// TIA Portal project "AUTO-5_UNLOADING_V15.1" (V15.1)

(* hardware
DEVICE "S7-1200 station_1"  S7-1200 Station
   slot 0: "Rack_0"  Rack  V1.0
   slot 1: "PLC_1"  CPU 1214C DC/DC/DC  6ES7 214-1AG40-0XB0  V4.2
   slot 2: "DI 16/DQ 16x24VDC_1"  6ES7 223-1BL32-0XB0  V2.0
   slot 3: "DI 16/DQ 16x24VDC_2"  6ES7 223-1BL32-0XB0  V2.0
DEVICE "HMI_1"  KTP700 Basic PN
   slot 0: "HMI_1"  KTP700 Basic PN  6AV2 123-2GB03-0AX0  15.1.0.0
   slot 1: "HMI_RT_1"  KTP700 Basic PN  6AV2 123-2GB03-0AX0  15.1.0.0
   slot 5: "HMI_1.IE_CP_1"  PROFINET Interface  15.0.1.0
      slot 1: "PROFINET Interface_1"  PROFINET Interface
         slot 1: "Port_1"  Port
DEVICE "GSD device"  GSD.Device.PN
   slot 0: "Rack"  Rack  V1.0
   slot 0: "CTEU-PN_1"  CTEU-PN  2201471  V1.0.0
      slot 0: "CTEU-PN"  CTEU-PN
      slot 1: "PN-IO Interface"  PN-IO Interface
         slot 1: "Port 1"  Port 1
         slot 2: "Port 2"  Port 2
   slot 1: "VAEM-L1-S-8-PT_1"  VAEM-L1-S-8-PT  573384
      slot 0: "VAEM-L1-S-8-PT"  VAEM-L1-S-8-PT
*)

// ===== PLC "PLC_1"  CPU 1214C DC/DC/DC =====

VAR_GLOBAL   // PLC tag table "Default tag table"
   "AUTO_ON_PB" AT %I0.6 : Bool;
   "AUTO_OFF_PB" AT %I0.7 : Bool;
   "CONTROL_OFF" AT %I0.1 : Bool;
   "AUTO_MODE" AT %I0.4 : Bool;
   "MANUAL_MODE" AT %I0.5 : Bool;
   "FAULT RESET" AT %I0.3 : Bool;
   "AIR PRESSURE SWITCH" AT %I1.1 : Bool;
   "PLUG_COUNT" AT %I1.2 : Bool;
   "Tag_14" AT %I1.3 : Bool;
   "Tag_15" AT %I1.4 : Bool;
   "Tag_16" AT %I1.5 : Bool;
   "Tag_17" AT %I2.0 : Bool;
   "Tag_19" AT %I2.2 : Bool;
   "INDIVIDULISER_DOWN" AT %I2.4 : Bool;
   "Tag_18" AT %I2.1 : Bool;
   "INDIVIDULISER_UP" AT %I2.3 : Bool;
   "TRAY LIFTING HEIGHT LEVELING_UP" AT %I2.5 : Bool;
   "TRAY LIFTING HEIGHT LEVELING_DOWN" AT %I2.6 : Bool;
   "TRAY LIFTING CYLINDER _UP" AT %I2.7 : Bool;
   "TRAY LIFTING CYLINDER _DOWN" AT %I3.0 : Bool;
   "TRAY LIFTING CYLINDER_FORWARD_RS" AT %I3.1 : Bool;
   "TRAY LIFTING CYLINDER_REVERSE_RS" AT %I3.2 : Bool;
   "PLUG LIFTING CYLINDER_UP" AT %I3.4 : Bool;
   "PLUG LIFTING CYLINDER_DOWN" AT %I3.3 : Bool;
   "PLUG LIFTING CYLINDER_FORWARD" AT %I3.5 : Bool;
   "PLUG LIFTING CYLINDER_REVERSE" AT %I3.6 : Bool;
   "TRAY STOPPER_UP" AT %I4.0 : Bool;
   "Tag_33" AT %I3.7 : Bool;
   "MPCB_TRIPPED" AT %I0.0 : Bool;
   "PLUG SENSOR MOUNTED ON CHUTE_INPUT" AT %I1.0 : Bool;
   "TRAY_PRESENT LEFT" AT %I4.7 : Bool;
   "TRAY RIGHT SENSOR" AT %I4.1 : Bool;
   "Tag_40" AT %I5.2 : Bool;
   "TRAY LEFT SENSOR" AT %I5.0 : Bool;
   "Tag_42" AT %I5.5 : Bool;
   "UPPER CONVEYOR LEFT  SENSOR" AT %I4.4 : Bool;
   "UPPER CONVEYOR RIGHT SENSOR" AT %I4.3 : Bool;
   "TRAY_PRESENT_RIGHT" AT %I4.5 : Bool;
   "WALKER BEAM UP" AT %Q0.0 : Bool;
   "WALKER BEAM DOWN" AT %Q0.1 : Bool;
   "Tag_12" AT %Q1.0 : Bool;
   "Tag_13" AT %Q1.1 : Bool;
   "CYCLE STRT ILPB INDICATOR" AT %Q0.3 : Bool;
   "PLUG_LIFT_DOWN" AT %Q6.0 : Bool;
   "PLUG LIFTING CYLINDER UP(1)" AT %Q6.1 : Bool;
   "GRIPPER_HOLD" AT %Q6.2 : Bool;
   "Tag_49" AT %Q7.4 : Bool;
   "TRAY PICKUP HEIGHT DOWN" AT %Q7.0 : Bool;
   "TRAY PICKUP UP" AT %Q7.1 : Bool;
   "TRAY LIFTING DOWN" AT %Q6.6 : Bool;
   "TRAY LIFTING CYLINDER  UP_OUTPUT" AT %Q6.7 : Bool;
   "TRAY LIFTING FWD_" AT %Q7.2 : Bool;
   "TRAY_LIFT_REVERSE" AT %Q7.3 : Bool;
   "PLUG_LIFT_REV" AT %Q6.4 : Bool;
   "PLUG_LIFT_FWD" AT %Q6.5 : Bool;
   "Tag_58" AT %Q7.6 : Bool;
   "Tag_59" AT %Q7.7 : Bool;
   "Tag_60" AT %Q7.5 : Bool;
   "AUTO CYCLE ON- YELLOW LAMP" AT %Q5.3 : Bool;
   "Tag_62" AT %Q5.4 : Bool;
   "ALL UNIT INITIAL- GREEN LAMP" AT %Q5.5 : Bool;
   "Tag_64" AT %Q0.6 : Bool;
   "FB_SENSOR OUTPUT" AT %Q5.6 : Bool;
   "RED LAMP" AT %Q5.7 : Bool;
   "GRIPPER_UNHOLD" AT %Q6.3 : Bool;
   "CONVEYOR -1 RUN FROM HMI" AT %M100.0 : Bool;
   "CONVEYOR -1 RUN OUTPUT" AT %M150.0 : Bool;
   "CONVEYOR 2 RUN FROM HMI" AT %M100.1 : Bool;
   "Tag_2" AT %M100.2 : Bool;
   "EMERGENCY" AT %M100.3 : Bool;
   "CYCLE START" AT %M100.4 : Bool;
   "CYCLE STOP" AT %M100.5 : Bool;
   "RESET" AT %M100.6 : Bool;
   "CONTROL ON" AT %M100.7 : Bool;
   "AUTO MODE" AT %M101.0 : Bool;
   "MANUAL MODE" AT %M101.1 : Bool;
   "AIR PRESSURE" AT %M101.2 : Bool;
   "PLUG SENSOR MOUNTED ON CHUTE" AT %M101.3 : Bool;
   "PLUG COUNTING" AT %M101.4 : Bool;
   "INDIVIDULISER-1 UP READ SWITCH" AT %M101.5 : Bool;
   "INDIVIDULISER-1 DOWN READ SWITCH" AT %M101.6 : Bool;
   "INDIVIDULISER -2 UP RS" AT %M101.7 : Bool;
   "INDIVIDULISER -2 DOWN RS" AT %M102.0 : Bool;
   "INDIVIDULISER -3 UP  RS" AT %M102.1 : Bool;
   "INDIVIDULISER -3 DOWN RS" AT %M102.2 : Bool;
   "INDIVIDULISER -4 UP RS" AT %M102.3 : Bool;
   "INDIVIDULISER -4 DOWN RS" AT %M102.4 : Bool;
   "TRAY LIFTING HEIGHT LEVELING UP READ SWITCH" AT %M102.5 : Bool;
   "TRAY LIFTING HEIGHT LEVELING DOWN READ SWITCH" AT %M102.6 : Bool;
   "TRAY LIFTING CYLINDER  UP  READ SWITCH" AT %M102.7 : Bool;
   "TRAY LIFTING CYLINDER DOWN READ SWITCH" AT %M103.0 : Bool;
   "TRAY LIFTING CYLINDER FORWARD READ SWITCH" AT %M103.1 : Bool;
   "TRAY LIFTING CYLINDER REVERSE READ SWITCH" AT %M103.2 : Bool;
   "PLUG LIFTING CYLINDER UP READ SWITCH" AT %M103.3 : Bool;
   "PLUG LIFTING CYLINDER DOWN READ SWITCH" AT %M103.4 : Bool;
   "PLUG LIFTING CYLINDER FORWARD READ SWITCH" AT %M103.5 : Bool;
   "PLUG LIFTING CYLINDER REVERSE READ SWITCH" AT %M103.6 : Bool;
   "TRAY STOPPER UP READ SWITCH" AT %M103.7 : Bool;
   "TRAY STOPPER DOWN READ SWITCH" AT %M104.0 : Bool;
   "TRAY LATCH UP READ SWITCH" AT %M104.1 : Bool;
   "TRAY LATCH DOWN READ SWITCH" AT %M104.2 : Bool;
   "CONVEYOR -1 MPCB TRIP" AT %M104.3 : Bool;
   "CONVEYOR -2 MPCB TRIP" AT %M104.4 : Bool;
   "INDIVIDUAL CYLINDER UP FROM HMI" AT %M104.5 : Bool;
   "INDIVIDUAL CYLINDER DOWN FROM HMI" AT %M104.6 : Bool;
   "TRAY LIFTING HEIGHT LEVELING UP FROM HMI" AT %M104.7 : Bool;
   "TRAY LIFTING HEIGHT LEVELING DOWN FROM HMI" AT %M105.0 : Bool;
   "TRAY LIFTING CYLINDER  UP FROM HMI" AT %M105.1 : Bool;
   "TRAY LIFTING CYLINDER  DOWN FROM HMI" AT %M105.2 : Bool;
   "TRAY LIFTING CYLINDER FORWARD FROM HMI" AT %M105.3 : Bool;
   "TRAY LIFTING CYLINDER REVERSE FROM HMI" AT %M105.4 : Bool;
   "PLUG LIFTING CYLINDER UP FROM HMI" AT %M105.5 : Bool;
   "PLUG LIFTING CYLINDER  DOWN FROM HMI" AT %M105.6 : Bool;
   "PLUG LIFTING CYLINDER FORWARD FROM HMI" AT %M105.7 : Bool;
   "CONVEYOR 2 RUN OUTPUT" AT %M150.1 : Bool;
   "INDIVIDULISER CYLINDER  UP" AT %M150.2 : Bool;
   "INDIVIDULISER CYLINDER DOWN" AT %M150.3 : Bool;
   "TRAY LIFTING HEIGHT LEVELING UP" AT %M150.4 : Bool;
   "TRAY LIFTING HEIGHT LEVELING DOWN" AT %M150.5 : Bool;
   "TRAY LIFTING CYLINDER  UP" AT %M150.6 : Bool;
   "TRAY LIFTING CYLINDER  DOWN" AT %M150.7 : Bool;
   "TRAY LIFTING CYLINDER FORWARD" AT %M151.0 : Bool;
   "TRAY LIFTING CYLINDER REVERSE" AT %M151.1 : Bool;
   "PLUG LIFTING CYLINDER UP" AT %M151.2 : Bool;
   "PLUG LIFTING CYLINDER DOWN" AT %M151.3 : Bool;
   "PLUG LIFTING CYLINDER FORWARD" AT %M151.4 : Bool;
   "PLUG LIFTING CYLINDER REVERSE" AT %M151.5 : Bool;
   "TRAY STOPPER UP" AT %M151.6 : Bool;
   "TRAY STOPPER DOWN" AT %M151.7 : Bool;
   "TRAY LATCH UP" AT %M152.0 : Bool;
   "TRAY LATCH DOWN" AT %M152.1 : Bool;
   "INITIAL CONDITION ON LAMP" AT %M152.2 : Bool;
   "TOWER LAMP RED" AT %M152.3 : Bool;
   "TOWER LAMP YELLOW" AT %M152.4 : Bool;
   "TOWER LAMP GREEN" AT %M152.5 : Bool;
   "BUZZER" AT %M152.6 : Bool;
   "PLUG LIFTING CYLINDER REVERSE FROM HMI" AT %M106.0 : Bool;
   "TRAY STOPPER UP FROM HMI" AT %M106.1 : Bool;
   "TRAY STOPPER DOWN FROM HMI" AT %M106.2 : Bool;
   "TRAY LATCH UP FROM HMI" AT %M106.3 : Bool;
   "TRAY LATCH DOWN FROM HMI" AT %M106.4 : Bool;
   "CYCLE START FLAG" AT %M200.0 : Bool;
   "ALL INDIVIDULISER UP RS" AT %M200.1 : Bool;
   "ALL INDIVIDULISER DOWN RS" AT %M200.2 : Bool;
   "Clock_Byte" AT %MB0 : Byte;
   "Clock_10Hz" AT %M0.0 : Bool;
   "Clock_5Hz" AT %M0.1 : Bool;
   "Clock_2.5Hz" AT %M0.2 : Bool;
   "Clock_2Hz" AT %M0.3 : Bool;
   "Clock_1.25Hz" AT %M0.4 : Bool;
   "Clock_1Hz" AT %M0.5 : Bool;
   "Clock_0.625Hz" AT %M0.6 : Bool;
   "Clock_0.5Hz" AT %M0.7 : Bool;
   "System_Byte" AT %MB1 : Byte;
   "FirstScan" AT %M1.0 : Bool;
   "DiagStatusUpdate" AT %M1.1 : Bool;
   "AlwaysTRUE" AT %M1.2 : Bool;
   "AlwaysFALSE" AT %M1.3 : Bool;
   "TRAY PRESENT SENSOR-LEFT PROXIMITY" AT %M106.5 : Bool;
   "TRAY PRESENT SENSOR-RIGHT PROXIMITY" AT %M106.6 : Bool;
   "TRAY PRESENT SENSOR BEFORE-LEFT PROXIMITY(1)" AT %M106.7 : Bool;
   "TRAY PRESENT BEFORE SENSOR-RIGHT PROXIMITY(1)" AT %M107.0 : Bool;
   "CONVEYOR -1 STOP FROM HMI" AT %M107.1 : Bool;
   "CONVEYOR -2 STOP FROM HMI" AT %M107.2 : Bool;
   "PLUG COUNTING PULSE" AT %M50.0 : Bool;
   "PLUG COUNTING RESET" AT %M50.1 : Bool;
   "Tag_36" AT %M30.0 : Bool;
   "TRAY LIFTING CYLINDER  DOWN_TRIGGER" AT %M30.1 : Bool;
   "Tag_43" AT %M25.0 : Bool;
   "Tag_44" AT %M20.0 : Bool;
   "Tag_46" AT %M10.1 : Bool;
   "TOWER LAMP BLUE" AT %M152.7 : Bool;
   "TOWER LAMP WHITE" AT %M153.0 : Bool;
   "PLUG HOLD FROM HMI" AT %M107.3 : Bool;
   "PLUD UNHOLD FROM HMI" AT %M107.4 : Bool;
   "PLUG HOLD O/P" AT %M153.1 : Bool;
   "PLUG UNHOLD O/P" AT %M153.2 : Bool;
   "TRIGGER_RESET_PLUG_COUNT" AT %M15.0 : Bool;
   "Tag_69" AT %M15.1 : Bool;
   "Tag_70" AT %M15.2 : Bool;
   "Tag_71" AT %M9.0 : Bool;
   "Tag_72" AT %M9.1 : Bool;
   "Tag_73" AT %M22.0 : Bool;
   "Tag_74" AT %M22.2 : Bool;
   "Tag_75" AT %M22.3 : Bool;
   "Tag_76" AT %M23.0 : Bool;
   "Tag_77" AT %M23.1 : Bool;
   "Tag_78" AT %M24.0 : Bool;
   "Tag_79" AT %M24.2 : Bool;
   "Tag_81" AT %M26.2 : Bool;
   "Tag_82" AT %M24.4 : Bool;
   "Tag_83" AT %M24.6 : Bool;
   "down tray present by pass on" AT %M25.5 : Bool;
   "delay 2s" AT %M40.0 : Bool;
   "1s delay for pallet sensors" AT %M40.2 : Bool;
   "DELAY 2S FOR DOWN FWD" AT %M40.4 : Bool;
   "Tag_84" AT %M99.0 : Bool;
   "DOWN B" AT %M90.1 : Bool;
   "Tag_41" AT %M90.2 : Bool;
   "Tag_47" AT %M90.7 : Bool;
   "UP B" AT %M90.5 : Bool;
   "INITIAL RESET" AT %I0.2 : Bool;
   "CONTROL ON OUTPUT" AT %Q0.7 : Bool;
   "Tag_7" AT %M15.5 : Bool;
   "Tag_39" AT %M16.3 : Bool;
   "Tag_85" AT %M16.5 : Bool;
   "INTER LOCK BIT TAKING UP/DOWN TRAY" AT %M17.2 : Bool;
   "Tag_87" AT %M17.4 : Bool;
   "Tag_1" AT %M16.1 : Bool;
   "Tag_3" AT %M16.2 : Bool;
   "PLUG PRESENT SENSOR AFTER REROLLING" AT %I5.4 : Bool;
   "AUTO WALKER UP" AT %M300.0 : Bool;
   "MAN WALKER UP" AT %M500.0 : Bool;
   "WALKER DOWN" AT %M300.1 : Bool;
   "MAN WALKER DOWN" AT %M500.1 : Bool;
   "Tag_5" AT %M300.2 : Bool;
   "HMI_PLUG_LIFT_UP" AT %M500.2 : Bool;
   "Tag_8" AT %M300.3 : Bool;
   "HMI_PLUG_LIFT_DOWN" AT %M500.3 : Bool;
   "Tag_10" AT %M300.4 : Bool;
   "HMI_GRIPPER_HOLD" AT %M500.4 : Bool;
   "Tag_21" AT %M300.5 : Bool;
   "HMI_GRIPPER_UNHOLD" AT %M500.5 : Bool;
   "Tag_23" AT %M300.6 : Bool;
   "HMI_TRAY_LIFT_DOWN" AT %M500.6 : Bool;
   "Tag_25" AT %M300.7 : Bool;
   "HMI_TRAY_LIFT_UP" AT %M500.7 : Bool;
   "Tag_27" AT %M301.0 : Bool;
   "HMI_TRAY_HEIGHT_DOWN" AT %M501.0 : Bool;
   "Tag_29" AT %M301.1 : Bool;
   "HMI_TRAY_HEIGHT_UP" AT %M501.1 : Bool;
   "Tag_31" AT %M301.2 : Bool;
   "HMI_TRAY_LIFT_FORWARD" AT %M501.2 : Bool;
   "Tag_34" AT %M301.3 : Bool;
   "HMI_TRAY_LIFT_REVERSE" AT %M501.3 : Bool;
   "AUTO ON" AT %M310.0 : Bool;
   "Tag_11" AT %M310.2 : Bool;
   "Tag_53" AT %M310.3 : Bool;
   "25 COUNT REACHED" AT %M310.5 : Bool;
   "Tag_86" AT %M310.7 : Bool;
   "ALL UNIT INITIAL" AT %M310.1 : Bool;
   "CONVY ON BIT" AT %M301.5 : Bool;
   "Tag_90" AT %M302.1 : Bool;
   "Tag_91" AT %M302.0 : Bool;
   "Tag_92" AT %MW300 : Int;
   "Tag_93" AT %MW302 : Int;
   "HMI_PLUG_LIFT_FWD" AT %M502.0 : Bool;
   "HMI_PLUG_LIFT_REV" AT %M502.1 : Bool;
   "Tag_96" AT %M312.0 : Bool;
   "PLUG LIFTING CYL DOWN SETBIT" AT %M600.3 : Bool;
   "PLUG GRIP SETBIT" AT %M600.4 : Bool;
   "Tag_99" AT %M610.5 : Bool;
   "TRAY UP SETBIT" AT %M610.0 : Bool;
   "Tag_101" AT %M610.2 : Bool;
   "PLUG GRIPPER UP CYL SETBIT" AT %M600.5 : Bool;
   "PLUG GRIP REV CYL SETBIT" AT %M600.6 : Bool;
   "PLUG LIFTING CYL DOWN  SETBIT" AT %M600.7 : Bool;
   "Tag_105" AT %M601.7 : Bool;
   "PLUG UNGRIP SETBIT" AT %M601.0 : Bool;
   "PLUG LIFTING UP CYL SETBIT" AT %M601.1 : Bool;
   "PLUG LIFTING FWD CYL SETBIT" AT %M601.2 : Bool;
   "Tag_109" AT %MW600 : Int;
   "Tag_110" AT %MW602 : Int;
   "Tag_111" AT %M610.4 : Bool;
   "Tag_112" AT %M610.6 : Bool;
   "TRAY FWD CYL SETBIT" AT %M611.0 : Bool;
   "TRAY DOWN CYL SETBIT" AT %M611.2 : Bool;
   "Tag_115" AT %M611.4 : Bool;
   "Tag_116" AT %M611.6 : Bool;
   "Tag_117" AT %M612.0 : Bool;
   "Tag_118" AT %M612.2 : Bool;
   "Tag_4" AT %MW604 : Int;
   "Tag_68" AT %MW606 : Int;
   "Tag_88" AT %MW610 : Int;
   "Tag_89" AT %MW612 : Int;
   "Tag_97" AT %M601.4 : Bool;
   "Tag_38" AT %M26.0 : Bool;
   "Tag_50" AT %M26.1 : Bool;
   "1s delay for pallet sensors_1" AT %M26.5 : Bool;
   "TRAY LIFTING HEIGHT LEVELING UP_TRIG" AT %M27.0 : Bool;
   "TRAY LIFT CYLINDER FORWARD TRIGGER" AT %M27.4 : Bool;
   "DELAY_2S_TIM" AT %M27.6 : Bool;
   "DELAY 2S FOR DOWN FWD_" AT %M27.7 : Bool;
   "Tag_51" AT %M28.0 : Bool;
   "TRAY LIFTING HEIGHT LEVELING DOWN_TRIGGER" AT %M28.1 : Bool;
   "TRAY LIFTING CYLINDER  UP_TRIGGER" AT %I30.0 : Bool;
   "TRAY LIFTING CYLINDER REVERSE_TRIGGER" AT %M31.0 : Bool;
   "PLUG_COUNT_DISPLAY" AT %MD32 : DInt;
   "SPARE" AT %Q0.5 : Bool;
   "ALL_UNIT_INITIAL" AT %Q0.2 : Bool;
   "Tag_6" AT %M613.0 : Bool;
   "Tag_9" AT %M163.0 : Bool;
   "Tag_20" AT %M163.1 : Bool;
   "Tag_22" AT %M613.1 : Bool;
   "Tag_24" AT %M613.2 : Bool;
   "parts full after rerolling" AT %I5.6 : Bool;
   "RELAY O/P" AT %Q2.0 : Bool;
   "RELAY TRIGGER BIT" AT %M613.6 : Bool;
   "Tag_26" AT %M614.0 : Bool;
   "Tag_28" AT %M614.1 : Bool;
   "ALARM_1" AT %MW60 : Word;
   "ALARM_2" AT %MW62 : Word;
   "Tag_30" AT %M60.0 : Bool;
   "CONTROL OFF" AT %M61.0 : Bool;
   "AUTO_OFF_ERROR" AT %M61.4 : Bool;
   "MPCB_TRIPPED_ERROR" AT %M61.3 : Bool;
   "AIR PRESSURE LOW ERROR" AT %M61.5 : Bool;
   "WAITING FOR PLUGS FROM SB UNIT ERROR" AT %M61.6 : Bool;
   "TRAY NOT  PRESENT ERROR" AT %M61.2 : Bool;
   "Tag_32" AT %M61.1 : Bool;
   "Tag_35" AT %M25.1 : Bool;
   "TRAY NOT PRESENT AT CONVEYOR END" AT %M61.7 : Bool;
   "Tag_45" AT %MW613 : Int;
   "Tag_48" AT %M630.0 : Bool;
   "INITIAL_SEQ_TRIGGER" AT %M110.0 : Bool;
   "TRAY_REVERSE_TRIGGER_INITIAL" AT %M110.1 : Bool;
   "TRAY_HEIGHT_UP_TRIG_INITIAL" AT %M110.2 : Bool;
   "TRAY HEIGHT FORWARD_TRIG_INITIAL" AT %M110.3 : Bool;
   "TRAY HEIGHT DOWN TRIG INITIAL" AT %M110.4 : Bool;
   "Tag_54" AT %MW110 : Int;
   "Tag_37" AT %M111.0 : Bool;
   "Tag_52" AT %M111.1 : Bool;
   "TRAY_HEIGHT_DOWN_INIT" AT %M111.3 : Bool;
   "Tag_55" AT %M112.0 : Bool;
   "Tag_56" AT %M112.1 : Bool;
   "Tag_57" AT %Q0.4 : Bool;
   "AUTO_OFF_TRIGGER_SINGLE CYCLE" AT %M112.2 : Bool;
   "Tag_63" AT %M113.0 : Bool;
   "PLUG TRANSFER SINGLE CYCLE TRIGGER" AT %M115.0 : Bool;
   "HMI_TRAY_PRESENT_INITIAL" AT %M25.2 : Bool;
   "TRAY HEIGHT LIFT INITIAL TRIGGER" AT %M116.0 : Bool;
   "TRAY _LIFT_REVERSE_INITIAL_TRIGGER" AT %M116.1 : Bool;
   "TRAY_LIFT_HEIGHT_DOWN_TRIGGER" AT %M116.2 : Bool;
   "TRAY_LIFT_FWD_INITIAL_TRIGGER" AT %M116.3 : Bool;
   "TRAY_LIFT_DOWN_INITIAL_TRIGGER" AT %M116.4 : Bool;
   "Tag_61" AT %MW115 : Int;
   "DUMMY" AT %M116.7 : Bool;
END_VAR

DATA_BLOCK "RETENTIVES"   // DB3
{ S7_Optimized_Access := 'FALSE' }
VERSION : 0.1
   VAR
      "PLUG COUNTER" : DInt;
      "RESET FLAG" : Bool;
      "PLUG FILLED" : Bool;
      "PLUG DATA" : DInt;
      "15 COUNTS REACH" : Bool;
      "PLUG LIFTING CYLINDER UP READ SWITCH" : Bool;
      "AUTO PLUG HOLD" : Bool;
      "AUTO PLUG UNHOLD" : Bool;
      "PLUG COUNTING RESET" : Bool;
      "ALL INDIVIDULISER DOWN CONFIRM" : Bool;
      "AUTO FWD FLag" : Bool;
      "AUTO REV FLAG" : Bool;
      "ALL INDIVIDULISER DOWN READ SWITCH" : Bool;
      "PLUG LIFTING CYLINDER UP" : Bool;
      "ERROR MSGS MOV BIT" : DInt;
      "ERROR FLAG ON" : Bool;
      "AUTO FWD FLAG DOWN" : Bool;
      "AUTO REV FLAG DOWN" : Bool;
      "AUTO FWD FLAG UP" : Bool;
      "AUTO REV FLAG UP" : Bool;
   END_VAR
BEGIN
END_DATA_BLOCK

// folder: System blocks/Program resources

DATA_BLOCK "PART PRESENT OFF DWELL"   // DB1
{ S7_Optimized_Access := 'TRUE' }
AUTHOR : Simatic
FAMILY : IEC
NAME : IEC_TMR
VERSION : 1.0
// stored: InstanceOfName IEC_TIMER
"IEC_TIMER"
BEGIN
END_DATA_BLOCK

DATA_BLOCK "PARTS COUNT"   // DB2
{ S7_Optimized_Access := 'TRUE' }
AUTHOR : Simatic
FAMILY : IEC
NAME : CNTR
VERSION : 1.0
// stored: InstanceOfName IEC_COUNTER
"IEC_COUNTER"
BEGIN
END_DATA_BLOCK

DATA_BLOCK "WALKER BEAM UP DWELL"   // DB4
{ S7_Optimized_Access := 'TRUE' }
AUTHOR : Simatic
FAMILY : IEC
NAME : IEC_TMR
VERSION : 1.0
// stored: InstanceOfName IEC_TIMER
"IEC_TIMER"
BEGIN
END_DATA_BLOCK

DATA_BLOCK "WALKER DOWN DWELL"   // DB5
{ S7_Optimized_Access := 'TRUE' }
AUTHOR : Simatic
FAMILY : IEC
NAME : IEC_TMR
VERSION : 1.0
// stored: InstanceOfName IEC_TIMER
"IEC_TIMER"
BEGIN
END_DATA_BLOCK

DATA_BLOCK "GRIP DWELL"   // DB6
{ S7_Optimized_Access := 'TRUE' }
AUTHOR : Simatic
FAMILY : IEC
NAME : IEC_TMR
VERSION : 1.0
// stored: InstanceOfName IEC_TIMER
"IEC_TIMER"
BEGIN
END_DATA_BLOCK

DATA_BLOCK "GRIPPER DOWN DWELL"   // DB7
{ S7_Optimized_Access := 'TRUE' }
AUTHOR : Simatic
FAMILY : IEC
NAME : IEC_TMR
VERSION : 1.0
// stored: InstanceOfName IEC_TIMER
"IEC_TIMER"
BEGIN
END_DATA_BLOCK

DATA_BLOCK "IEC_Timer_0_DB_6"   // DB8
{ S7_Optimized_Access := 'TRUE' }
AUTHOR : Simatic
FAMILY : IEC
NAME : IEC_TMR
VERSION : 1.0
// stored: InstanceOfName IEC_TIMER
"IEC_TIMER"
BEGIN
END_DATA_BLOCK

DATA_BLOCK "IEC_Timer_0_DB_5"   // DB9
{ S7_Optimized_Access := 'TRUE' }
AUTHOR : Simatic
FAMILY : IEC
NAME : IEC_TMR
VERSION : 1.0
// stored: InstanceOfName IEC_TIMER
"IEC_TIMER"
BEGIN
END_DATA_BLOCK

DATA_BLOCK "UNGRIP DWELL"   // DB10
{ S7_Optimized_Access := 'TRUE' }
AUTHOR : Simatic
FAMILY : IEC
NAME : IEC_TMR
VERSION : 1.0
// stored: InstanceOfName IEC_TIMER
"IEC_TIMER"
BEGIN
END_DATA_BLOCK

DATA_BLOCK "DOWN DWELL"   // DB11
{ S7_Optimized_Access := 'TRUE' }
AUTHOR : Simatic
FAMILY : IEC
NAME : IEC_TMR
VERSION : 1.0
// stored: InstanceOfName IEC_TIMER
"IEC_TIMER"
BEGIN
END_DATA_BLOCK

DATA_BLOCK "IEC_Timer_0_DB"   // DB12
{ S7_Optimized_Access := 'TRUE' }
AUTHOR : Simatic
FAMILY : IEC
NAME : IEC_TMR
VERSION : 1.0
// stored: InstanceOfName IEC_TIMER
"IEC_TIMER"
BEGIN
END_DATA_BLOCK

DATA_BLOCK "IEC_Timer_0_DB_1"   // DB13
{ S7_Optimized_Access := 'TRUE' }
AUTHOR : Simatic
FAMILY : IEC
NAME : IEC_TMR
VERSION : 1.0
// stored: InstanceOfName IEC_TIMER
"IEC_TIMER"
BEGIN
END_DATA_BLOCK

DATA_BLOCK "IEC_Timer_0_DB_2"   // DB14
{ S7_Optimized_Access := 'TRUE' }
AUTHOR : Simatic
FAMILY : IEC
NAME : IEC_TMR
VERSION : 1.0
// stored: InstanceOfName IEC_TIMER
"IEC_TIMER"
BEGIN
END_DATA_BLOCK

DATA_BLOCK "IEC_Timer_0_DB_3"   // DB15
{ S7_Optimized_Access := 'TRUE' }
AUTHOR : Simatic
FAMILY : IEC
NAME : IEC_TMR
VERSION : 1.0
// stored: InstanceOfName IEC_TIMER
"IEC_TIMER"
BEGIN
END_DATA_BLOCK

DATA_BLOCK "IEC_Timer_0_DB_7"   // DB16
{ S7_Optimized_Access := 'TRUE' }
AUTHOR : Simatic
FAMILY : IEC
NAME : IEC_TMR
VERSION : 1.0
// stored: InstanceOfName IEC_TIMER
"IEC_TIMER"
BEGIN
END_DATA_BLOCK

DATA_BLOCK "IEC_Timer_0_DB_4"   // DB17
{ S7_Optimized_Access := 'TRUE' }
AUTHOR : Simatic
FAMILY : IEC
NAME : IEC_TMR
VERSION : 1.0
// stored: InstanceOfName IEC_TIMER
"IEC_TIMER"
BEGIN
END_DATA_BLOCK

DATA_BLOCK "TRAY ABSENT AT LIFTING SIDE"   // DB18
{ S7_Optimized_Access := 'TRUE' }
AUTHOR : Simatic
FAMILY : IEC
NAME : IEC_TMR
VERSION : 1.0
// stored: InstanceOfName IEC_TIMER
"IEC_TIMER"
BEGIN
END_DATA_BLOCK

DATA_BLOCK "time delay"   // DB19
{ S7_Optimized_Access := 'TRUE' }
AUTHOR : Simatic
FAMILY : IEC
NAME : IEC_TMR
VERSION : 1.0
// stored: InstanceOfName IEC_TIMER
"IEC_TIMER"
BEGIN
END_DATA_BLOCK

DATA_BLOCK "Time delay after plug present"   // DB21
{ S7_Optimized_Access := 'TRUE' }
AUTHOR : Simatic
FAMILY : IEC
NAME : IEC_TMR
VERSION : 1.0
// stored: InstanceOfName IEC_TIMER
"IEC_TIMER"
BEGIN
END_DATA_BLOCK

// folder: (top level)

FUNCTION "INITIAL SEQUENCE" : Void   // FC1, LAD
{ S7_Optimized_Access := 'TRUE' }
VERSION : 0.1
   VAR_TEMP   // added for the SCL form of the ladder/FBD networks
      _w1 : Bool;
   END_VAR
BEGIN

REGION Network 1: TRAY INITIAL SEQUENCE
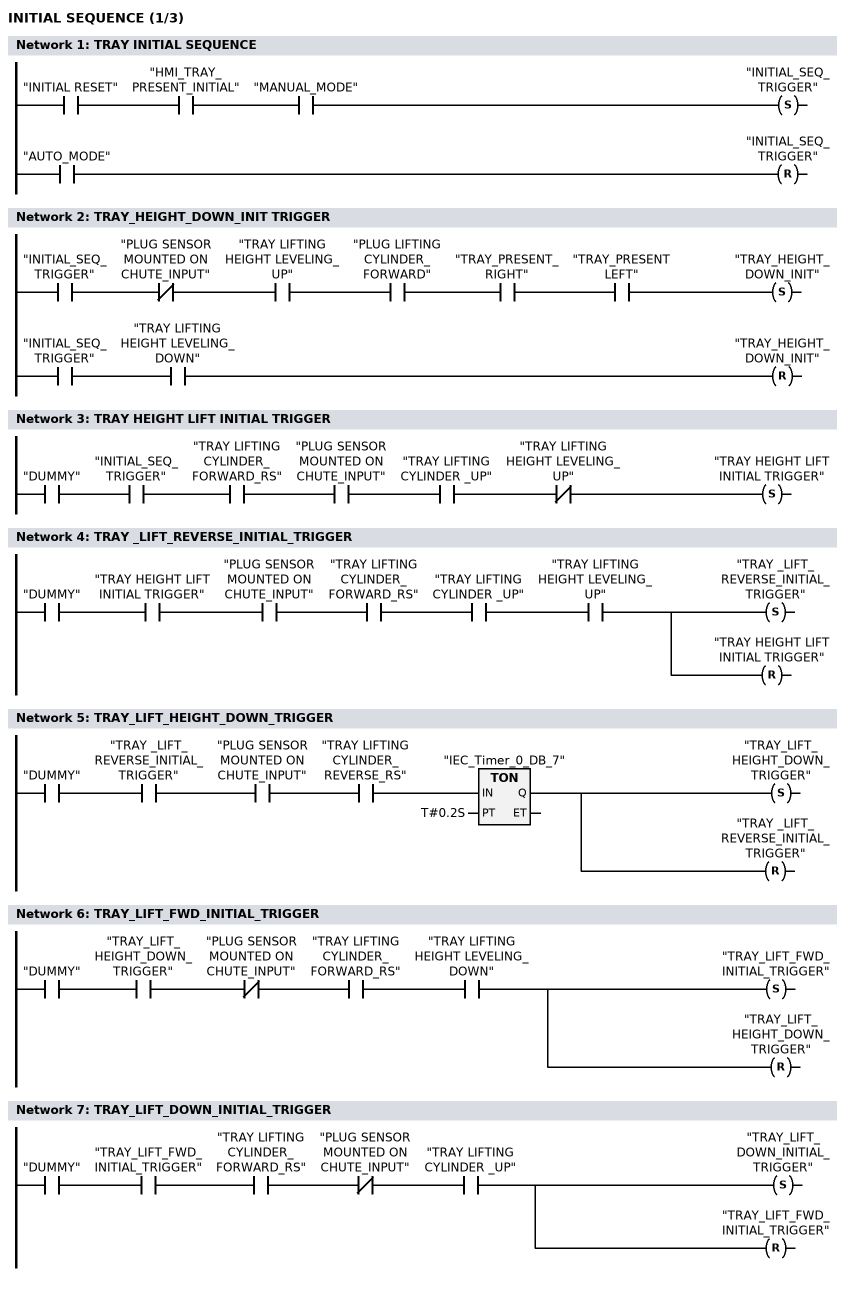
   RUNG wire#powerrail
      Contact( "INITIAL RESET" )
      Contact( "HMI_TRAY_PRESENT_INITIAL" )
      Contact( "MANUAL_MODE" )
      S_Coil( "INITIAL_SEQ_TRIGGER" )
   END_RUNG
   RUNG wire#powerrail
      Contact( "AUTO_MODE" )
      R_Coil( "INITIAL_SEQ_TRIGGER" )
   END_RUNG
   // the same network as SCL:
   IF "INITIAL RESET" AND "HMI_TRAY_PRESENT_INITIAL" AND "MANUAL_MODE" THEN
       "INITIAL_SEQ_TRIGGER" := TRUE;
   END_IF;
   IF "AUTO_MODE" THEN "INITIAL_SEQ_TRIGGER" := FALSE; END_IF;
END_REGION

REGION Network 2: TRAY_HEIGHT_DOWN_INIT TRIGGER
   RUNG wire#powerrail
      Contact( "INITIAL_SEQ_TRIGGER" )
      I_Contact( "PLUG SENSOR MOUNTED ON CHUTE_INPUT" )
      Contact( "TRAY LIFTING HEIGHT LEVELING_UP" )
      Contact( "PLUG LIFTING CYLINDER_FORWARD" )
      Contact( "TRAY_PRESENT_RIGHT" )
      Contact( "TRAY_PRESENT LEFT" )
      S_Coil( "TRAY_HEIGHT_DOWN_INIT" )
   END_RUNG
   RUNG wire#powerrail
      Contact( "INITIAL_SEQ_TRIGGER" )
      Contact( "TRAY LIFTING HEIGHT LEVELING_DOWN" )
      R_Coil( "TRAY_HEIGHT_DOWN_INIT" )
   END_RUNG
   // the same network as SCL:
   IF "INITIAL_SEQ_TRIGGER" AND NOT "PLUG SENSOR MOUNTED ON CHUTE_INPUT" AND "TRAY LIFTING HEIGHT LEVELING_UP" AND "PLUG LIFTING CYLINDER_FORWARD" AND "TRAY_PRESENT_RIGHT" AND "TRAY_PRESENT LEFT" THEN
       "TRAY_HEIGHT_DOWN_INIT" := TRUE;
   END_IF;
   IF "INITIAL_SEQ_TRIGGER" AND "TRAY LIFTING HEIGHT LEVELING_DOWN" THEN
       "TRAY_HEIGHT_DOWN_INIT" := FALSE;
   END_IF;
END_REGION

REGION Network 3: TRAY HEIGHT LIFT INITIAL TRIGGER
   RUNG wire#powerrail
      Contact( "DUMMY" )
      Contact( "INITIAL_SEQ_TRIGGER" )
      Contact( "TRAY LIFTING CYLINDER_FORWARD_RS" )
      Contact( "PLUG SENSOR MOUNTED ON CHUTE_INPUT" )
      Contact( "TRAY LIFTING CYLINDER _UP" )
      I_Contact( "TRAY LIFTING HEIGHT LEVELING_UP" )
      S_Coil( "TRAY HEIGHT LIFT INITIAL TRIGGER" )
   END_RUNG
   // the same network as SCL:
   IF "DUMMY" AND "INITIAL_SEQ_TRIGGER" AND "TRAY LIFTING CYLINDER_FORWARD_RS" AND "PLUG SENSOR MOUNTED ON CHUTE_INPUT" AND "TRAY LIFTING CYLINDER _UP" AND NOT "TRAY LIFTING HEIGHT LEVELING_UP" THEN
       "TRAY HEIGHT LIFT INITIAL TRIGGER" := TRUE;
   END_IF;
END_REGION

REGION Network 4: TRAY _LIFT_REVERSE_INITIAL_TRIGGER
   RUNG wire#powerrail
      Contact( "DUMMY" )
      Contact( "TRAY HEIGHT LIFT INITIAL TRIGGER" )
      Contact( "PLUG SENSOR MOUNTED ON CHUTE_INPUT" )
      Contact( "TRAY LIFTING CYLINDER_FORWARD_RS" )
      Contact( "TRAY LIFTING CYLINDER _UP" )
      Contact( "TRAY LIFTING HEIGHT LEVELING_UP" )
      wire#w1
      S_Coil( "TRAY _LIFT_REVERSE_INITIAL_TRIGGER" )
   END_RUNG
   RUNG wire#w1
      R_Coil( "TRAY HEIGHT LIFT INITIAL TRIGGER" )
   END_RUNG
   // the same network as SCL:
   IF "DUMMY" AND "TRAY HEIGHT LIFT INITIAL TRIGGER" AND "PLUG SENSOR MOUNTED ON CHUTE_INPUT" AND "TRAY LIFTING CYLINDER_FORWARD_RS" AND "TRAY LIFTING CYLINDER _UP" AND "TRAY LIFTING HEIGHT LEVELING_UP" THEN
       "TRAY _LIFT_REVERSE_INITIAL_TRIGGER" := TRUE;
       "TRAY HEIGHT LIFT INITIAL TRIGGER" := FALSE;
   END_IF;
END_REGION

REGION Network 5: TRAY_LIFT_HEIGHT_DOWN_TRIGGER
   "IEC_Timer_0_DB_7".TON(IN := "DUMMY" AND "TRAY _LIFT_REVERSE_INITIAL_TRIGGER" AND "PLUG SENSOR MOUNTED ON CHUTE_INPUT" AND "TRAY LIFTING CYLINDER_REVERSE_RS",
                          PT := T#0.2S);
   IF "IEC_Timer_0_DB_7".Q THEN
       "TRAY_LIFT_HEIGHT_DOWN_TRIGGER" := TRUE;
       "TRAY _LIFT_REVERSE_INITIAL_TRIGGER" := FALSE;
   END_IF;
END_REGION

REGION Network 6: TRAY_LIFT_FWD_INITIAL_TRIGGER
   RUNG wire#powerrail
      Contact( "DUMMY" )
      Contact( "TRAY_LIFT_HEIGHT_DOWN_TRIGGER" )
      I_Contact( "PLUG SENSOR MOUNTED ON CHUTE_INPUT" )
      Contact( "TRAY LIFTING CYLINDER_FORWARD_RS" )
      Contact( "TRAY LIFTING HEIGHT LEVELING_DOWN" )
      wire#w1
      S_Coil( "TRAY_LIFT_FWD_INITIAL_TRIGGER" )
   END_RUNG
   RUNG wire#w1
      R_Coil( "TRAY_LIFT_HEIGHT_DOWN_TRIGGER" )
   END_RUNG
   // the same network as SCL:
   IF "DUMMY" AND "TRAY_LIFT_HEIGHT_DOWN_TRIGGER" AND NOT "PLUG SENSOR MOUNTED ON CHUTE_INPUT" AND "TRAY LIFTING CYLINDER_FORWARD_RS" AND "TRAY LIFTING HEIGHT LEVELING_DOWN" THEN
       "TRAY_LIFT_FWD_INITIAL_TRIGGER" := TRUE;
       "TRAY_LIFT_HEIGHT_DOWN_TRIGGER" := FALSE;
   END_IF;
END_REGION

REGION Network 7: TRAY_LIFT_DOWN_INITIAL_TRIGGER
   RUNG wire#powerrail
      Contact( "DUMMY" )
      Contact( "TRAY_LIFT_FWD_INITIAL_TRIGGER" )
      Contact( "TRAY LIFTING CYLINDER_FORWARD_RS" )
      I_Contact( "PLUG SENSOR MOUNTED ON CHUTE_INPUT" )
      Contact( "TRAY LIFTING CYLINDER _UP" )
      wire#w1
      S_Coil( "TRAY_LIFT_DOWN_INITIAL_TRIGGER" )
   END_RUNG
   RUNG wire#w1
      R_Coil( "TRAY_LIFT_FWD_INITIAL_TRIGGER" )
   END_RUNG
   // the same network as SCL:
   IF "DUMMY" AND "TRAY_LIFT_FWD_INITIAL_TRIGGER" AND "TRAY LIFTING CYLINDER_FORWARD_RS" AND NOT "PLUG SENSOR MOUNTED ON CHUTE_INPUT" AND "TRAY LIFTING CYLINDER _UP" THEN
       "TRAY_LIFT_DOWN_INITIAL_TRIGGER" := TRUE;
       "TRAY_LIFT_FWD_INITIAL_TRIGGER" := FALSE;
   END_IF;
END_REGION

REGION Network 8
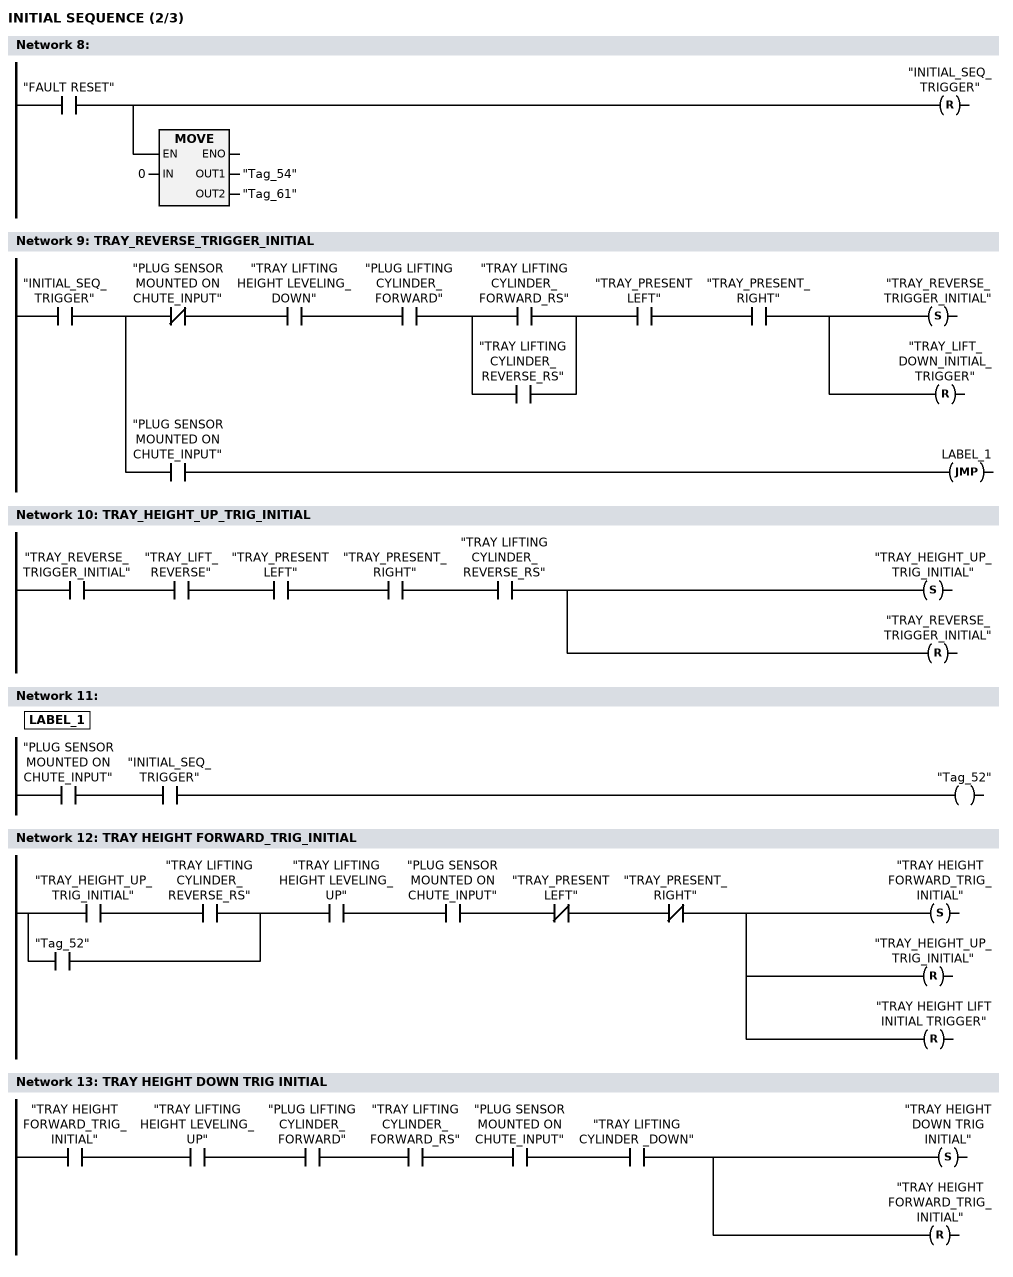
   RUNG wire#powerrail
      Contact( "FAULT RESET" )
      wire#w1
      R_Coil( "INITIAL_SEQ_TRIGGER" )
   END_RUNG
   RUNG wire#w1
      Move(in := 0, out1 => "Tag_54", out2 => "Tag_61")
   END_RUNG
   // the same network as SCL:
   IF "FAULT RESET" THEN
       "INITIAL_SEQ_TRIGGER" := FALSE;
       "Tag_54" := 0;
       "Tag_61" := 0;
   END_IF;
END_REGION

REGION Network 9: TRAY_REVERSE_TRIGGER_INITIAL
   RUNG wire#powerrail
      Contact( "INITIAL_SEQ_TRIGGER" )
      wire#w1
      I_Contact( "PLUG SENSOR MOUNTED ON CHUTE_INPUT" )
      Contact( "TRAY LIFTING HEIGHT LEVELING_DOWN" )
      Contact( "PLUG LIFTING CYLINDER_FORWARD" )
      wire#w2
      Contact( "TRAY LIFTING CYLINDER_FORWARD_RS" )
      wire#w3
      Contact( "TRAY_PRESENT LEFT" )
      Contact( "TRAY_PRESENT_RIGHT" )
      wire#w4
      S_Coil( "TRAY_REVERSE_TRIGGER_INITIAL" )
   END_RUNG
   RUNG wire#w2
      Contact( "TRAY LIFTING CYLINDER_REVERSE_RS" )
   END_RUNG wire#w3
   RUNG wire#w4
      R_Coil( "TRAY_LIFT_DOWN_INITIAL_TRIGGER" )
   END_RUNG
   RUNG wire#w1
      Contact( "PLUG SENSOR MOUNTED ON CHUTE_INPUT" )
      JumpCoil( LABEL_1 )
   END_RUNG
   // the same network as SCL:
   IF "INITIAL_SEQ_TRIGGER" AND NOT "PLUG SENSOR MOUNTED ON CHUTE_INPUT" AND "TRAY LIFTING HEIGHT LEVELING_DOWN" AND "PLUG LIFTING CYLINDER_FORWARD" AND ("TRAY LIFTING CYLINDER_FORWARD_RS" OR "TRAY LIFTING CYLINDER_REVERSE_RS") AND "TRAY_PRESENT LEFT" AND "TRAY_PRESENT_RIGHT" THEN
       "TRAY_REVERSE_TRIGGER_INITIAL" := TRUE;
       "TRAY_LIFT_DOWN_INITIAL_TRIGGER" := FALSE;
   END_IF;
   IF "INITIAL_SEQ_TRIGGER" AND "PLUG SENSOR MOUNTED ON CHUTE_INPUT" THEN GOTO LABEL_1; END_IF;
END_REGION

REGION Network 10: TRAY_HEIGHT_UP_TRIG_INITIAL
   RUNG wire#powerrail
      Contact( "TRAY_REVERSE_TRIGGER_INITIAL" )
      Contact( "TRAY_LIFT_REVERSE" )
      Contact( "TRAY_PRESENT LEFT" )
      Contact( "TRAY_PRESENT_RIGHT" )
      Contact( "TRAY LIFTING CYLINDER_REVERSE_RS" )
      wire#w1
      S_Coil( "TRAY_HEIGHT_UP_TRIG_INITIAL" )
   END_RUNG
   RUNG wire#w1
      R_Coil( "TRAY_REVERSE_TRIGGER_INITIAL" )
   END_RUNG
   // the same network as SCL:
   IF "TRAY_REVERSE_TRIGGER_INITIAL" AND "TRAY_LIFT_REVERSE" AND "TRAY_PRESENT LEFT" AND "TRAY_PRESENT_RIGHT" AND "TRAY LIFTING CYLINDER_REVERSE_RS" THEN
       "TRAY_HEIGHT_UP_TRIG_INITIAL" := TRUE;
       "TRAY_REVERSE_TRIGGER_INITIAL" := FALSE;
   END_IF;
END_REGION

REGION Network 11
   Label( LABEL_1 )
   RUNG wire#powerrail
      Contact( "PLUG SENSOR MOUNTED ON CHUTE_INPUT" )
      Contact( "INITIAL_SEQ_TRIGGER" )
      Coil( "Tag_52" )
   END_RUNG
   // the same network as SCL:
   LABEL_1:
   "Tag_52" := "PLUG SENSOR MOUNTED ON CHUTE_INPUT" AND "INITIAL_SEQ_TRIGGER";
END_REGION

REGION Network 12: TRAY HEIGHT FORWARD_TRIG_INITIAL
   RUNG wire#powerrail
      Contact( "TRAY_HEIGHT_UP_TRIG_INITIAL" )
      Contact( "TRAY LIFTING CYLINDER_REVERSE_RS" )
      wire#w1
      Contact( "TRAY LIFTING HEIGHT LEVELING_UP" )
      Contact( "PLUG SENSOR MOUNTED ON CHUTE_INPUT" )
      I_Contact( "TRAY_PRESENT LEFT" )
      I_Contact( "TRAY_PRESENT_RIGHT" )
      wire#w2
      S_Coil( "TRAY HEIGHT FORWARD_TRIG_INITIAL" )
   END_RUNG
   RUNG wire#powerrail
      Contact( "Tag_52" )
   END_RUNG wire#w1
   RUNG wire#w2
      R_Coil( "TRAY_HEIGHT_UP_TRIG_INITIAL" )
   END_RUNG
   RUNG wire#w2
      R_Coil( "TRAY HEIGHT LIFT INITIAL TRIGGER" )
   END_RUNG
   // the same network as SCL:
   IF (("TRAY_HEIGHT_UP_TRIG_INITIAL" AND "TRAY LIFTING CYLINDER_REVERSE_RS") OR "Tag_52") AND "TRAY LIFTING HEIGHT LEVELING_UP" AND "PLUG SENSOR MOUNTED ON CHUTE_INPUT" AND NOT "TRAY_PRESENT LEFT" AND NOT "TRAY_PRESENT_RIGHT" THEN
       "TRAY HEIGHT FORWARD_TRIG_INITIAL" := TRUE;
   END_IF;
   #_w1 := (("TRAY_HEIGHT_UP_TRIG_INITIAL" AND "TRAY LIFTING CYLINDER_REVERSE_RS") OR "Tag_52") AND "TRAY LIFTING HEIGHT LEVELING_UP" AND "PLUG SENSOR MOUNTED ON CHUTE_INPUT" AND NOT "TRAY_PRESENT LEFT" AND NOT "TRAY_PRESENT_RIGHT";
   IF #_w1 THEN
       "TRAY_HEIGHT_UP_TRIG_INITIAL" := FALSE;
       "TRAY HEIGHT LIFT INITIAL TRIGGER" := FALSE;
   END_IF;
END_REGION

REGION Network 13: TRAY HEIGHT DOWN TRIG INITIAL
   RUNG wire#powerrail
      Contact( "TRAY HEIGHT FORWARD_TRIG_INITIAL" )
      Contact( "TRAY LIFTING HEIGHT LEVELING_UP" )
      Contact( "PLUG LIFTING CYLINDER_FORWARD" )
      Contact( "TRAY LIFTING CYLINDER_FORWARD_RS" )
      Contact( "PLUG SENSOR MOUNTED ON CHUTE_INPUT" )
      Contact( "TRAY LIFTING CYLINDER _DOWN" )
      wire#w1
      S_Coil( "TRAY HEIGHT DOWN TRIG INITIAL" )
   END_RUNG
   RUNG wire#w1
      R_Coil( "TRAY HEIGHT FORWARD_TRIG_INITIAL" )
   END_RUNG
   // the same network as SCL:
   IF "TRAY HEIGHT FORWARD_TRIG_INITIAL" AND "TRAY LIFTING HEIGHT LEVELING_UP" AND "PLUG LIFTING CYLINDER_FORWARD" AND "TRAY LIFTING CYLINDER_FORWARD_RS" AND "PLUG SENSOR MOUNTED ON CHUTE_INPUT" AND "TRAY LIFTING CYLINDER _DOWN" THEN
       "TRAY HEIGHT DOWN TRIG INITIAL" := TRUE;
       "TRAY HEIGHT FORWARD_TRIG_INITIAL" := FALSE;
   END_IF;
END_REGION

REGION Network 14
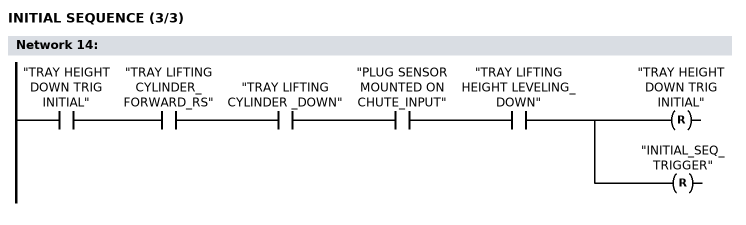
   RUNG wire#powerrail
      Contact( "TRAY HEIGHT DOWN TRIG INITIAL" )
      Contact( "TRAY LIFTING CYLINDER_FORWARD_RS" )
      Contact( "TRAY LIFTING CYLINDER _DOWN" )
      Contact( "PLUG SENSOR MOUNTED ON CHUTE_INPUT" )
      Contact( "TRAY LIFTING HEIGHT LEVELING_DOWN" )
      wire#w1
      R_Coil( "TRAY HEIGHT DOWN TRIG INITIAL" )
   END_RUNG
   RUNG wire#w1
      R_Coil( "INITIAL_SEQ_TRIGGER" )
   END_RUNG
   // the same network as SCL:
   #_w1 := "TRAY HEIGHT DOWN TRIG INITIAL" AND "TRAY LIFTING CYLINDER_FORWARD_RS" AND "TRAY LIFTING CYLINDER _DOWN" AND "PLUG SENSOR MOUNTED ON CHUTE_INPUT" AND "TRAY LIFTING HEIGHT LEVELING_DOWN";
   IF #_w1 THEN
       "TRAY HEIGHT DOWN TRIG INITIAL" := FALSE;
       "INITIAL_SEQ_TRIGGER" := FALSE;
   END_IF;
END_REGION
END_FUNCTION

FUNCTION "ALARMS" : Void   // FC2, LAD
{ S7_Optimized_Access := 'TRUE' }
VERSION : 0.1
   VAR_TEMP   // added for the SCL form of the ladder/FBD networks
      _w1 : Bool;
      _w2 : Bool;
   END_VAR
BEGIN

REGION Network 1: CONTROL OFF ALARM
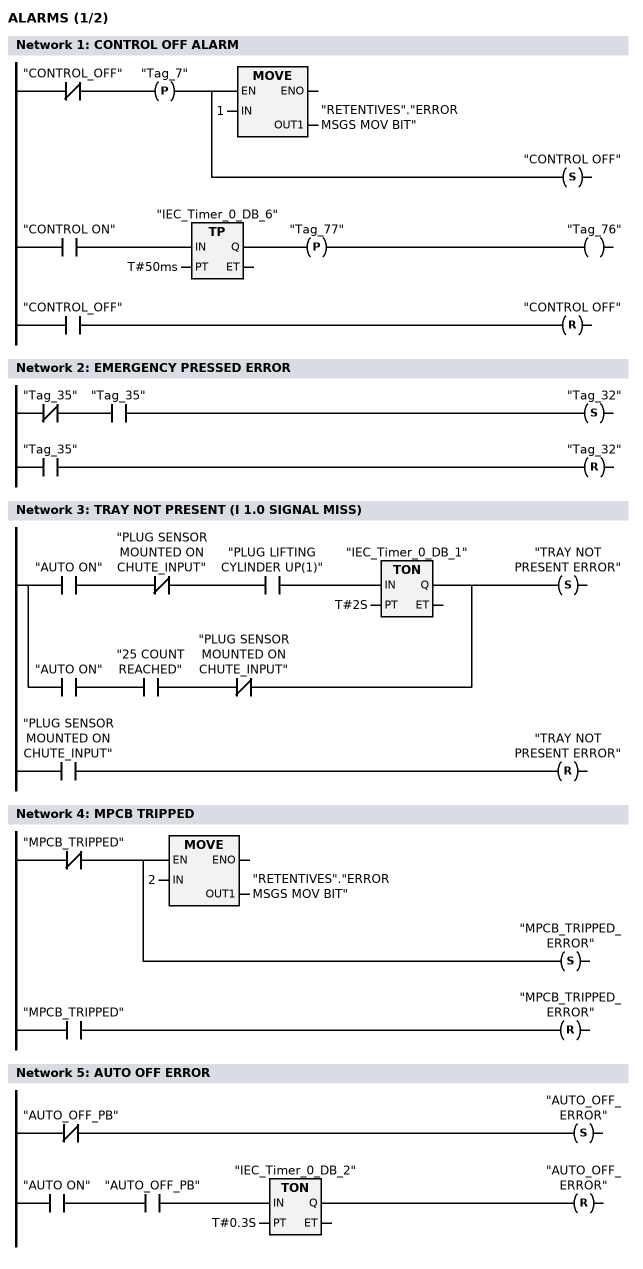
   #_w1 := NOT "CONTROL_OFF" AND NOT "Tag_7";   // rising edge
   "Tag_7" := NOT "CONTROL_OFF";
   IF #_w1 THEN
       "RETENTIVES"."ERROR MSGS MOV BIT" := 1;
       "CONTROL OFF" := TRUE;
   END_IF;
   "IEC_Timer_0_DB_6".TP(IN := "CONTROL ON", PT := T#50ms);
   #_w2 := "IEC_Timer_0_DB_6".Q AND NOT "Tag_77";   // rising edge
   "Tag_77" := "IEC_Timer_0_DB_6".Q;
   "Tag_76" := #_w2;
   IF "CONTROL_OFF" THEN "CONTROL OFF" := FALSE; END_IF;
END_REGION

REGION Network 2: EMERGENCY PRESSED ERROR
   RUNG wire#powerrail
      I_Contact( "Tag_35" )
      Contact( "Tag_35" )
      S_Coil( "Tag_32" )
   END_RUNG
   RUNG wire#powerrail
      Contact( "Tag_35" )
      R_Coil( "Tag_32" )
   END_RUNG
   // the same network as SCL:
   IF NOT "Tag_35" AND "Tag_35" THEN "Tag_32" := TRUE; END_IF;
   IF "Tag_35" THEN "Tag_32" := FALSE; END_IF;
END_REGION

REGION Network 3: TRAY NOT PRESENT (I 1.0 SIGNAL MISS)
   "IEC_Timer_0_DB_1".TON(IN := "AUTO ON" AND NOT "PLUG SENSOR MOUNTED ON CHUTE_INPUT" AND "PLUG LIFTING CYLINDER UP(1)",
                          PT := T#2S);
   IF "IEC_Timer_0_DB_1".Q OR ("AUTO ON" AND "25 COUNT REACHED" AND NOT "PLUG SENSOR MOUNTED ON CHUTE_INPUT") THEN
       "TRAY NOT  PRESENT ERROR" := TRUE;
   END_IF;
   IF "PLUG SENSOR MOUNTED ON CHUTE_INPUT" THEN "TRAY NOT  PRESENT ERROR" := FALSE; END_IF;
END_REGION

REGION Network 4: MPCB TRIPPED
   RUNG wire#powerrail
      I_Contact( "MPCB_TRIPPED" )
      wire#w1
      Move(in := 2, out1 => "RETENTIVES"."ERROR MSGS MOV BIT")
   END_RUNG
   RUNG wire#w1
      S_Coil( "MPCB_TRIPPED_ERROR" )
   END_RUNG
   RUNG wire#powerrail
      Contact( "MPCB_TRIPPED" )
      R_Coil( "MPCB_TRIPPED_ERROR" )
   END_RUNG
   // the same network as SCL:
   IF NOT "MPCB_TRIPPED" THEN
       "RETENTIVES"."ERROR MSGS MOV BIT" := 2;
       "MPCB_TRIPPED_ERROR" := TRUE;
   END_IF;
   IF "MPCB_TRIPPED" THEN "MPCB_TRIPPED_ERROR" := FALSE; END_IF;
END_REGION

REGION Network 5: AUTO OFF ERROR
   IF NOT "AUTO_OFF_PB" THEN "AUTO_OFF_ERROR" := TRUE; END_IF;
   "IEC_Timer_0_DB_2".TON(IN := "AUTO ON" AND "AUTO_OFF_PB", PT := T#0.3S);
   IF "IEC_Timer_0_DB_2".Q THEN "AUTO_OFF_ERROR" := FALSE; END_IF;
END_REGION

REGION Network 6: PNEUMATIC AIR PRESSURE LOW
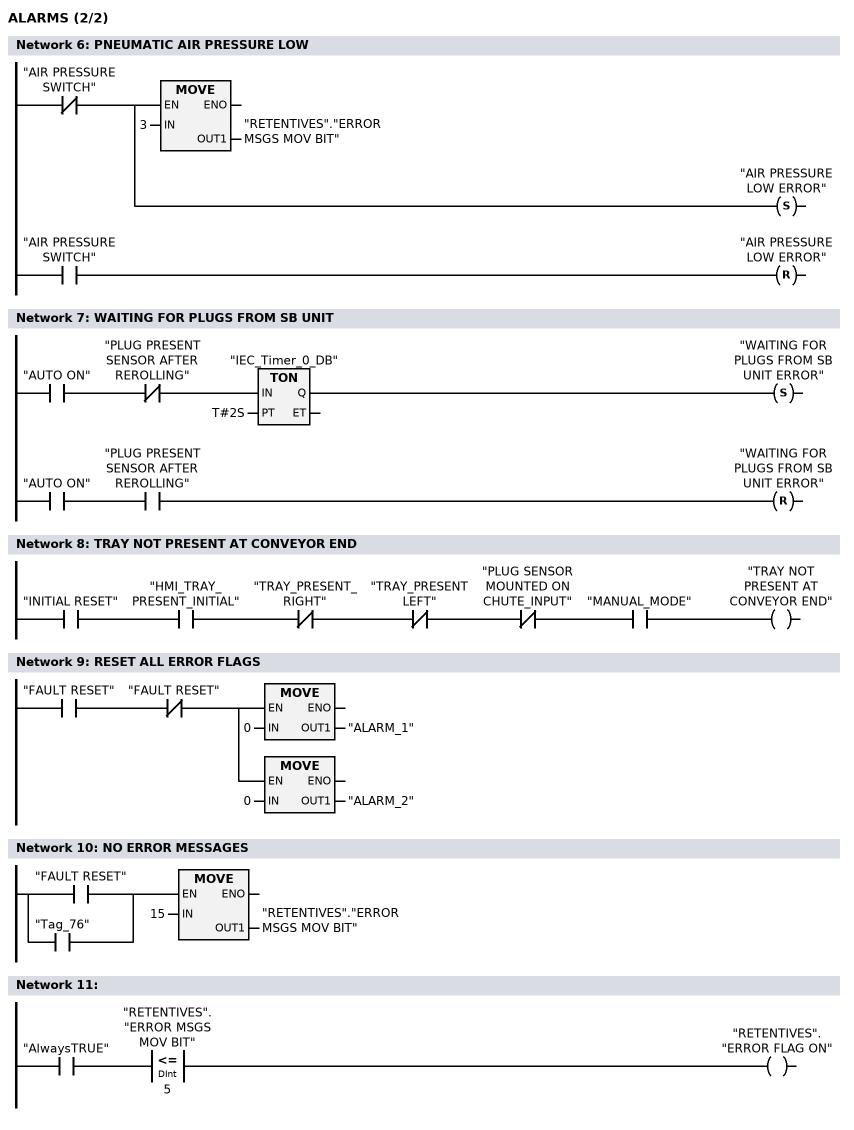
   RUNG wire#powerrail
      I_Contact( "AIR PRESSURE SWITCH" )
      wire#w1
      Move(in := 3, out1 => "RETENTIVES"."ERROR MSGS MOV BIT")
   END_RUNG
   RUNG wire#w1
      S_Coil( "AIR PRESSURE LOW ERROR" )
   END_RUNG
   RUNG wire#powerrail
      Contact( "AIR PRESSURE SWITCH" )
      R_Coil( "AIR PRESSURE LOW ERROR" )
   END_RUNG
   // the same network as SCL:
   IF NOT "AIR PRESSURE SWITCH" THEN
       "RETENTIVES"."ERROR MSGS MOV BIT" := 3;
       "AIR PRESSURE LOW ERROR" := TRUE;
   END_IF;
   IF "AIR PRESSURE SWITCH" THEN "AIR PRESSURE LOW ERROR" := FALSE; END_IF;
END_REGION

REGION Network 7: WAITING FOR PLUGS FROM SB UNIT
   "IEC_Timer_0_DB".TON(IN := "AUTO ON" AND NOT "PLUG PRESENT SENSOR AFTER REROLLING", PT := T#2S);
   IF "IEC_Timer_0_DB".Q THEN "WAITING FOR PLUGS FROM SB UNIT ERROR" := TRUE; END_IF;
   IF "AUTO ON" AND "PLUG PRESENT SENSOR AFTER REROLLING" THEN
       "WAITING FOR PLUGS FROM SB UNIT ERROR" := FALSE;
   END_IF;
END_REGION

REGION Network 8: TRAY NOT PRESENT AT CONVEYOR END
   RUNG wire#powerrail
      Contact( "INITIAL RESET" )
      Contact( "HMI_TRAY_PRESENT_INITIAL" )
      I_Contact( "TRAY_PRESENT_RIGHT" )
      I_Contact( "TRAY_PRESENT LEFT" )
      I_Contact( "PLUG SENSOR MOUNTED ON CHUTE_INPUT" )
      Contact( "MANUAL_MODE" )
      Coil( "TRAY NOT PRESENT AT CONVEYOR END" )
   END_RUNG
   // the same network as SCL:
   "TRAY NOT PRESENT AT CONVEYOR END" := "INITIAL RESET" AND "HMI_TRAY_PRESENT_INITIAL" AND NOT "TRAY_PRESENT_RIGHT" AND NOT "TRAY_PRESENT LEFT" AND NOT "PLUG SENSOR MOUNTED ON CHUTE_INPUT" AND "MANUAL_MODE";
END_REGION

REGION Network 9: RESET ALL ERROR FLAGS
   RUNG wire#powerrail
      Contact( "FAULT RESET" )
      I_Contact( "FAULT RESET" )
      wire#w1
      Move(in := 0, out1 => "ALARM_1")
   END_RUNG
   RUNG wire#w1
      Move(in := 0, out1 => "ALARM_2")
   END_RUNG
   // the same network as SCL:
   IF "FAULT RESET" AND NOT "FAULT RESET" THEN
       "ALARM_1" := 0;
       "ALARM_2" := 0;
   END_IF;
END_REGION

REGION Network 10: NO ERROR MESSAGES
   RUNG wire#powerrail
      Contact( "FAULT RESET" )
      wire#w1
      Move(in := 15, out1 => "RETENTIVES"."ERROR MSGS MOV BIT")
   END_RUNG
   RUNG wire#powerrail
      Contact( "Tag_76" )
   END_RUNG wire#w1
   // the same network as SCL:
   IF "FAULT RESET" OR "Tag_76" THEN "RETENTIVES"."ERROR MSGS MOV BIT" := 15; END_IF;
END_REGION

REGION Network 11
   RUNG wire#powerrail
      Contact( "AlwaysTRUE" )
      { S7_Templates := "SrcType := DInt" } LE_Contact(in1 := "RETENTIVES"."ERROR MSGS MOV BIT", in2 := 5)
      Coil( "RETENTIVES"."ERROR FLAG ON" )
   END_RUNG
   // the same network as SCL:
   "RETENTIVES"."ERROR FLAG ON" := "AlwaysTRUE" AND ("RETENTIVES"."ERROR MSGS MOV BIT" <= 5);
END_REGION
END_FUNCTION

FUNCTION "CONTROL ON LAMPS" : Void   // FC3, LAD
{ S7_Optimized_Access := 'FALSE' }
VERSION : 0.1
BEGIN

REGION Network 1: CYCLE START
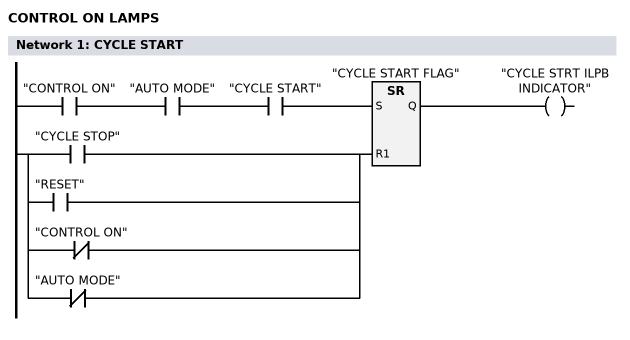
   RUNG wire#powerrail
      Contact( "CONTROL ON" )
      Contact( "AUTO MODE" )
      Contact( "CYCLE START" )
      S_SR(operand := "CYCLE START FLAG", r1 := wire#w1)
      Coil( "CYCLE STRT ILPB INDICATOR" )
   END_RUNG
   RUNG wire#powerrail
      Contact( "CYCLE STOP" )
   END_RUNG wire#w1
   RUNG wire#powerrail
      Contact( "RESET" )
   END_RUNG wire#w1
   RUNG wire#powerrail
      I_Contact( "CONTROL ON" )
   END_RUNG wire#w1
   RUNG wire#powerrail
      I_Contact( "AUTO MODE" )
   END_RUNG wire#w1
   // the same network as SCL:
   IF "CONTROL ON" AND "AUTO MODE" AND "CYCLE START" THEN
       "CYCLE START FLAG" := TRUE;   // SR flip-flop
   END_IF;
   IF "CYCLE STOP" OR "RESET" OR NOT "CONTROL ON" OR NOT "AUTO MODE" THEN
       "CYCLE START FLAG" := FALSE;
   END_IF;
   "CYCLE STRT ILPB INDICATOR" := "CYCLE START FLAG";
END_REGION
END_FUNCTION

FUNCTION "NEW OUTPUT BLOCK" : Void   // FC6, LAD
{ S7_Optimized_Access := 'TRUE' }
VERSION : 0.1
BEGIN

REGION Network 1: WALKER BEAM UP
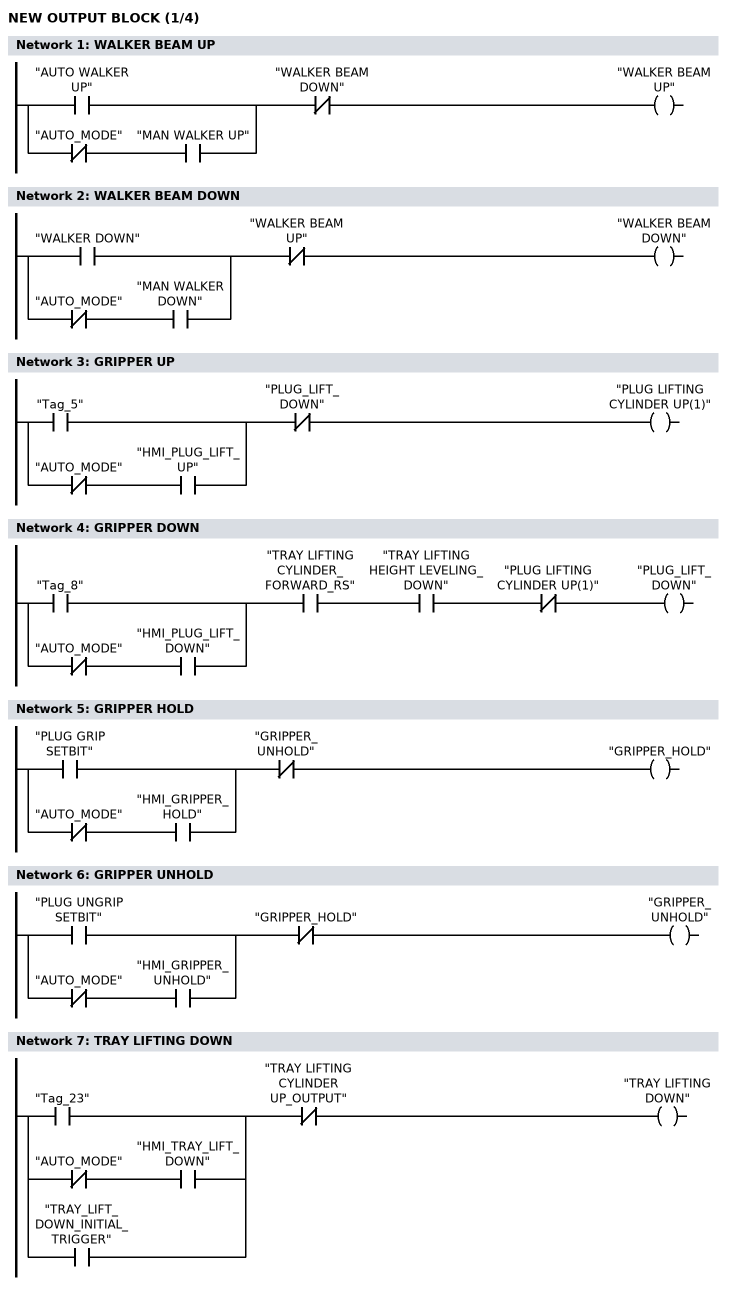
   RUNG wire#powerrail
      Contact( "AUTO WALKER UP" )
      wire#w1
      I_Contact( "WALKER BEAM DOWN" )
      Coil( "WALKER BEAM UP" )
   END_RUNG
   RUNG wire#powerrail
      I_Contact( "AUTO_MODE" )
      Contact( "MAN WALKER UP" )
   END_RUNG wire#w1
   // the same network as SCL:
   "WALKER BEAM UP" := ("AUTO WALKER UP" OR (NOT "AUTO_MODE" AND "MAN WALKER UP")) AND NOT "WALKER BEAM DOWN";
END_REGION

REGION Network 2: WALKER BEAM DOWN
   RUNG wire#powerrail
      Contact( "WALKER DOWN" )
      wire#w1
      I_Contact( "WALKER BEAM UP" )
      Coil( "WALKER BEAM DOWN" )
   END_RUNG
   RUNG wire#powerrail
      I_Contact( "AUTO_MODE" )
      Contact( "MAN WALKER DOWN" )
   END_RUNG wire#w1
   // the same network as SCL:
   "WALKER BEAM DOWN" := ("WALKER DOWN" OR (NOT "AUTO_MODE" AND "MAN WALKER DOWN")) AND NOT "WALKER BEAM UP";
END_REGION

REGION Network 3: GRIPPER UP
   RUNG wire#powerrail
      Contact( "Tag_5" )
      wire#w1
      I_Contact( "PLUG_LIFT_DOWN" )
      Coil( "PLUG LIFTING CYLINDER UP(1)" )
   END_RUNG
   RUNG wire#powerrail
      I_Contact( "AUTO_MODE" )
      Contact( "HMI_PLUG_LIFT_UP" )
   END_RUNG wire#w1
   // the same network as SCL:
   "PLUG LIFTING CYLINDER UP(1)" := ("Tag_5" OR (NOT "AUTO_MODE" AND "HMI_PLUG_LIFT_UP")) AND NOT "PLUG_LIFT_DOWN";
END_REGION

REGION Network 4: GRIPPER DOWN
   RUNG wire#powerrail
      Contact( "Tag_8" )
      wire#w1
      Contact( "TRAY LIFTING CYLINDER_FORWARD_RS" )
      Contact( "TRAY LIFTING HEIGHT LEVELING_DOWN" )
      I_Contact( "PLUG LIFTING CYLINDER UP(1)" )
      Coil( "PLUG_LIFT_DOWN" )
   END_RUNG
   RUNG wire#powerrail
      I_Contact( "AUTO_MODE" )
      Contact( "HMI_PLUG_LIFT_DOWN" )
   END_RUNG wire#w1
   // the same network as SCL:
   "PLUG_LIFT_DOWN" := ("Tag_8" OR (NOT "AUTO_MODE" AND "HMI_PLUG_LIFT_DOWN")) AND "TRAY LIFTING CYLINDER_FORWARD_RS" AND "TRAY LIFTING HEIGHT LEVELING_DOWN" AND NOT "PLUG LIFTING CYLINDER UP(1)";
END_REGION

REGION Network 5: GRIPPER HOLD
   RUNG wire#powerrail
      Contact( "PLUG GRIP SETBIT" )
      wire#w1
      I_Contact( "GRIPPER_UNHOLD" )
      Coil( "GRIPPER_HOLD" )
   END_RUNG
   RUNG wire#powerrail
      I_Contact( "AUTO_MODE" )
      Contact( "HMI_GRIPPER_HOLD" )
   END_RUNG wire#w1
   // the same network as SCL:
   "GRIPPER_HOLD" := ("PLUG GRIP SETBIT" OR (NOT "AUTO_MODE" AND "HMI_GRIPPER_HOLD")) AND NOT "GRIPPER_UNHOLD";
END_REGION

REGION Network 6: GRIPPER UNHOLD
   RUNG wire#powerrail
      Contact( "PLUG UNGRIP SETBIT" )
      wire#w1
      I_Contact( "GRIPPER_HOLD" )
      Coil( "GRIPPER_UNHOLD" )
   END_RUNG
   RUNG wire#powerrail
      I_Contact( "AUTO_MODE" )
      Contact( "HMI_GRIPPER_UNHOLD" )
   END_RUNG wire#w1
   // the same network as SCL:
   "GRIPPER_UNHOLD" := ("PLUG UNGRIP SETBIT" OR (NOT "AUTO_MODE" AND "HMI_GRIPPER_UNHOLD")) AND NOT "GRIPPER_HOLD";
END_REGION

REGION Network 7: TRAY LIFTING DOWN
   RUNG wire#powerrail
      Contact( "Tag_23" )
      wire#w1
      I_Contact( "TRAY LIFTING CYLINDER  UP_OUTPUT" )
      Coil( "TRAY LIFTING DOWN" )
   END_RUNG
   RUNG wire#powerrail
      I_Contact( "AUTO_MODE" )
      Contact( "HMI_TRAY_LIFT_DOWN" )
   END_RUNG wire#w1
   RUNG wire#powerrail
      Contact( "TRAY_LIFT_DOWN_INITIAL_TRIGGER" )
   END_RUNG wire#w1
   // the same network as SCL:
   "TRAY LIFTING DOWN" := ("Tag_23" OR (NOT "AUTO_MODE" AND "HMI_TRAY_LIFT_DOWN") OR "TRAY_LIFT_DOWN_INITIAL_TRIGGER") AND NOT "TRAY LIFTING CYLINDER  UP_OUTPUT";
END_REGION

REGION Network 8: TRAY LIFTING CYLINDER UP
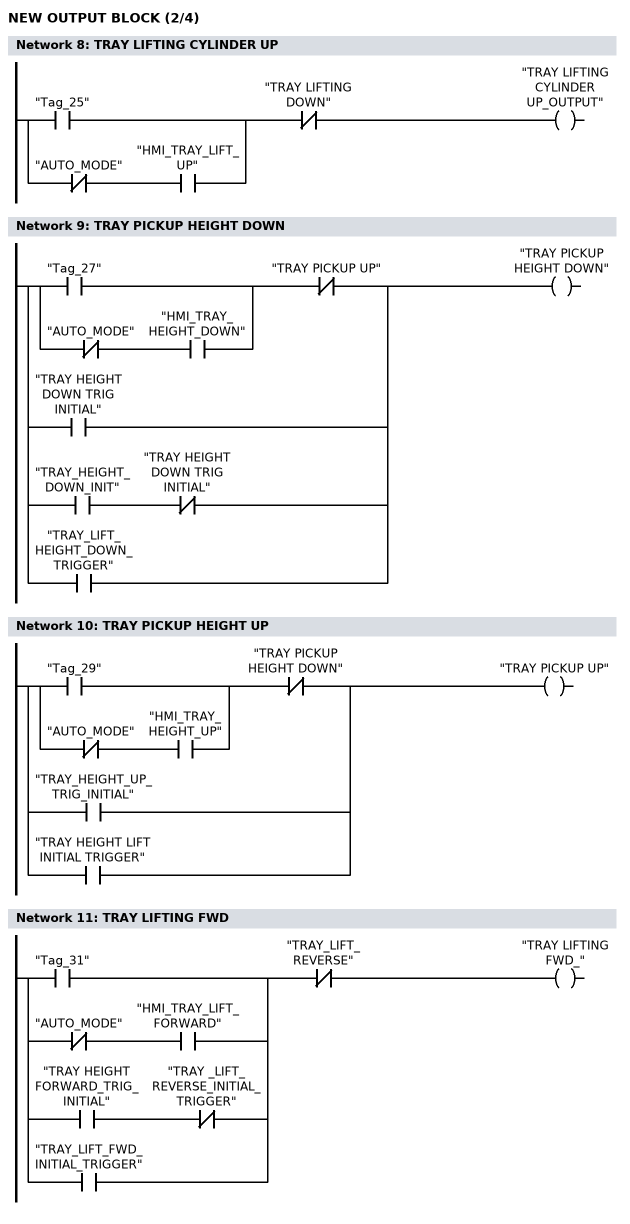
   RUNG wire#powerrail
      Contact( "Tag_25" )
      wire#w1
      I_Contact( "TRAY LIFTING DOWN" )
      Coil( "TRAY LIFTING CYLINDER  UP_OUTPUT" )
   END_RUNG
   RUNG wire#powerrail
      I_Contact( "AUTO_MODE" )
      Contact( "HMI_TRAY_LIFT_UP" )
   END_RUNG wire#w1
   // the same network as SCL:
   "TRAY LIFTING CYLINDER  UP_OUTPUT" := ("Tag_25" OR (NOT "AUTO_MODE" AND "HMI_TRAY_LIFT_UP")) AND NOT "TRAY LIFTING DOWN";
END_REGION

REGION Network 9: TRAY PICKUP HEIGHT DOWN
   RUNG wire#powerrail
      Contact( "Tag_27" )
      wire#w1
      I_Contact( "TRAY PICKUP UP" )
      wire#w2
      Coil( "TRAY PICKUP HEIGHT DOWN" )
   END_RUNG
   RUNG wire#powerrail
      I_Contact( "AUTO_MODE" )
      Contact( "HMI_TRAY_HEIGHT_DOWN" )
   END_RUNG wire#w1
   RUNG wire#powerrail
      Contact( "TRAY HEIGHT DOWN TRIG INITIAL" )
   END_RUNG wire#w2
   RUNG wire#powerrail
      Contact( "TRAY_HEIGHT_DOWN_INIT" )
      I_Contact( "TRAY HEIGHT DOWN TRIG INITIAL" )
   END_RUNG wire#w2
   RUNG wire#powerrail
      Contact( "TRAY_LIFT_HEIGHT_DOWN_TRIGGER" )
   END_RUNG wire#w2
   // the same network as SCL:
   "TRAY PICKUP HEIGHT DOWN" := (("Tag_27" OR (NOT "AUTO_MODE" AND "HMI_TRAY_HEIGHT_DOWN")) AND NOT "TRAY PICKUP UP") OR "TRAY HEIGHT DOWN TRIG INITIAL" OR ("TRAY_HEIGHT_DOWN_INIT" AND NOT "TRAY HEIGHT DOWN TRIG INITIAL") OR "TRAY_LIFT_HEIGHT_DOWN_TRIGGER";
END_REGION

REGION Network 10: TRAY PICKUP HEIGHT UP
   RUNG wire#powerrail
      Contact( "Tag_29" )
      wire#w1
      I_Contact( "TRAY PICKUP HEIGHT DOWN" )
      wire#w2
      Coil( "TRAY PICKUP UP" )
   END_RUNG
   RUNG wire#powerrail
      I_Contact( "AUTO_MODE" )
      Contact( "HMI_TRAY_HEIGHT_UP" )
   END_RUNG wire#w1
   RUNG wire#powerrail
      Contact( "TRAY_HEIGHT_UP_TRIG_INITIAL" )
   END_RUNG wire#w2
   RUNG wire#powerrail
      Contact( "TRAY HEIGHT LIFT INITIAL TRIGGER" )
   END_RUNG wire#w2
   // the same network as SCL:
   "TRAY PICKUP UP" := (("Tag_29" OR (NOT "AUTO_MODE" AND "HMI_TRAY_HEIGHT_UP")) AND NOT "TRAY PICKUP HEIGHT DOWN") OR "TRAY_HEIGHT_UP_TRIG_INITIAL" OR "TRAY HEIGHT LIFT INITIAL TRIGGER";
END_REGION

REGION Network 11: TRAY LIFTING FWD
   RUNG wire#powerrail
      Contact( "Tag_31" )
      wire#w1
      I_Contact( "TRAY_LIFT_REVERSE" )
      Coil( "TRAY LIFTING FWD_" )
   END_RUNG
   RUNG wire#powerrail
      I_Contact( "AUTO_MODE" )
      Contact( "HMI_TRAY_LIFT_FORWARD" )
   END_RUNG wire#w1
   RUNG wire#powerrail
      Contact( "TRAY HEIGHT FORWARD_TRIG_INITIAL" )
      I_Contact( "TRAY _LIFT_REVERSE_INITIAL_TRIGGER" )
   END_RUNG wire#w1
   RUNG wire#powerrail
      Contact( "TRAY_LIFT_FWD_INITIAL_TRIGGER" )
   END_RUNG wire#w1
   // the same network as SCL:
   "TRAY LIFTING FWD_" := ("Tag_31" OR (NOT "AUTO_MODE" AND "HMI_TRAY_LIFT_FORWARD") OR ("TRAY HEIGHT FORWARD_TRIG_INITIAL" AND NOT "TRAY _LIFT_REVERSE_INITIAL_TRIGGER") OR "TRAY_LIFT_FWD_INITIAL_TRIGGER") AND NOT "TRAY_LIFT_REVERSE";
END_REGION

REGION Network 12: TRAY LIFTING REV
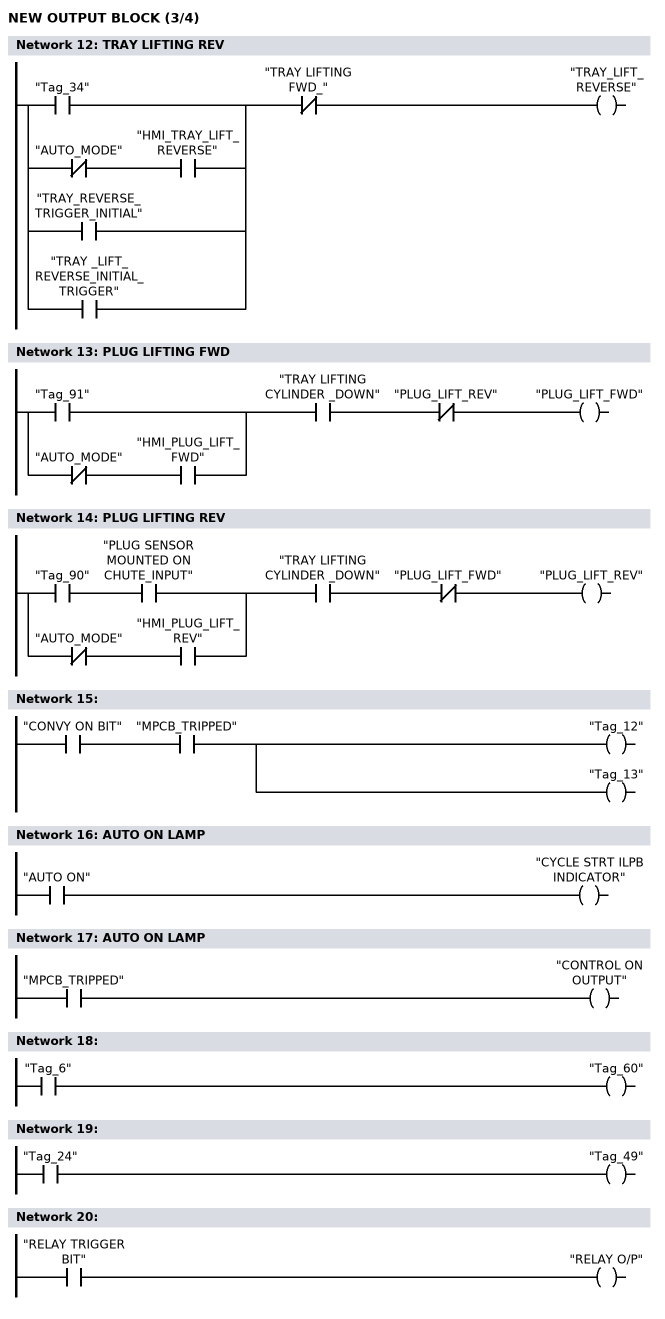
   RUNG wire#powerrail
      Contact( "Tag_34" )
      wire#w1
      I_Contact( "TRAY LIFTING FWD_" )
      Coil( "TRAY_LIFT_REVERSE" )
   END_RUNG
   RUNG wire#powerrail
      I_Contact( "AUTO_MODE" )
      Contact( "HMI_TRAY_LIFT_REVERSE" )
   END_RUNG wire#w1
   RUNG wire#powerrail
      Contact( "TRAY_REVERSE_TRIGGER_INITIAL" )
   END_RUNG wire#w1
   RUNG wire#powerrail
      Contact( "TRAY _LIFT_REVERSE_INITIAL_TRIGGER" )
   END_RUNG wire#w1
   // the same network as SCL:
   "TRAY_LIFT_REVERSE" := ("Tag_34" OR (NOT "AUTO_MODE" AND "HMI_TRAY_LIFT_REVERSE") OR "TRAY_REVERSE_TRIGGER_INITIAL" OR "TRAY _LIFT_REVERSE_INITIAL_TRIGGER") AND NOT "TRAY LIFTING FWD_";
END_REGION

REGION Network 13: PLUG LIFTING FWD
   RUNG wire#powerrail
      Contact( "Tag_91" )
      wire#w1
      Contact( "TRAY LIFTING CYLINDER _DOWN" )
      I_Contact( "PLUG_LIFT_REV" )
      Coil( "PLUG_LIFT_FWD" )
   END_RUNG
   RUNG wire#powerrail
      I_Contact( "AUTO_MODE" )
      Contact( "HMI_PLUG_LIFT_FWD" )
   END_RUNG wire#w1
   // the same network as SCL:
   "PLUG_LIFT_FWD" := ("Tag_91" OR (NOT "AUTO_MODE" AND "HMI_PLUG_LIFT_FWD")) AND "TRAY LIFTING CYLINDER _DOWN" AND NOT "PLUG_LIFT_REV";
END_REGION

REGION Network 14: PLUG LIFTING REV
   RUNG wire#powerrail
      Contact( "Tag_90" )
      Contact( "PLUG SENSOR MOUNTED ON CHUTE_INPUT" )
      wire#w1
      Contact( "TRAY LIFTING CYLINDER _DOWN" )
      I_Contact( "PLUG_LIFT_FWD" )
      Coil( "PLUG_LIFT_REV" )
   END_RUNG
   RUNG wire#powerrail
      I_Contact( "AUTO_MODE" )
      Contact( "HMI_PLUG_LIFT_REV" )
   END_RUNG wire#w1
   // the same network as SCL:
   "PLUG_LIFT_REV" := (("Tag_90" AND "PLUG SENSOR MOUNTED ON CHUTE_INPUT") OR (NOT "AUTO_MODE" AND "HMI_PLUG_LIFT_REV")) AND "TRAY LIFTING CYLINDER _DOWN" AND NOT "PLUG_LIFT_FWD";
END_REGION

REGION Network 15
   RUNG wire#powerrail
      Contact( "CONVY ON BIT" )
      Contact( "MPCB_TRIPPED" )
      wire#w1
      Coil( "Tag_12" )
   END_RUNG
   RUNG wire#w1
      Coil( "Tag_13" )
   END_RUNG
   // the same network as SCL:
   "Tag_12" := "CONVY ON BIT" AND "MPCB_TRIPPED";
   "Tag_13" := "Tag_12";
END_REGION

REGION Network 16: AUTO ON LAMP
   RUNG wire#powerrail
      Contact( "AUTO ON" )
      Coil( "CYCLE STRT ILPB INDICATOR" )
   END_RUNG
   // the same network as SCL:
   "CYCLE STRT ILPB INDICATOR" := "AUTO ON";
END_REGION

REGION Network 17: AUTO ON LAMP
   RUNG wire#powerrail
      Contact( "MPCB_TRIPPED" )
      Coil( "CONTROL ON OUTPUT" )
   END_RUNG
   // the same network as SCL:
   "CONTROL ON OUTPUT" := "MPCB_TRIPPED";
END_REGION

REGION Network 18
   RUNG wire#powerrail
      Contact( "Tag_6" )
      Coil( "Tag_60" )
   END_RUNG
   // the same network as SCL:
   "Tag_60" := "Tag_6";
END_REGION

REGION Network 19
   RUNG wire#powerrail
      Contact( "Tag_24" )
      Coil( "Tag_49" )
   END_RUNG
   // the same network as SCL:
   "Tag_49" := "Tag_24";
END_REGION

REGION Network 20
   RUNG wire#powerrail
      Contact( "RELAY TRIGGER BIT" )
      Coil( "RELAY O/P" )
   END_RUNG
   // the same network as SCL:
   "RELAY O/P" := "RELAY TRIGGER BIT";
END_REGION

REGION Network 21
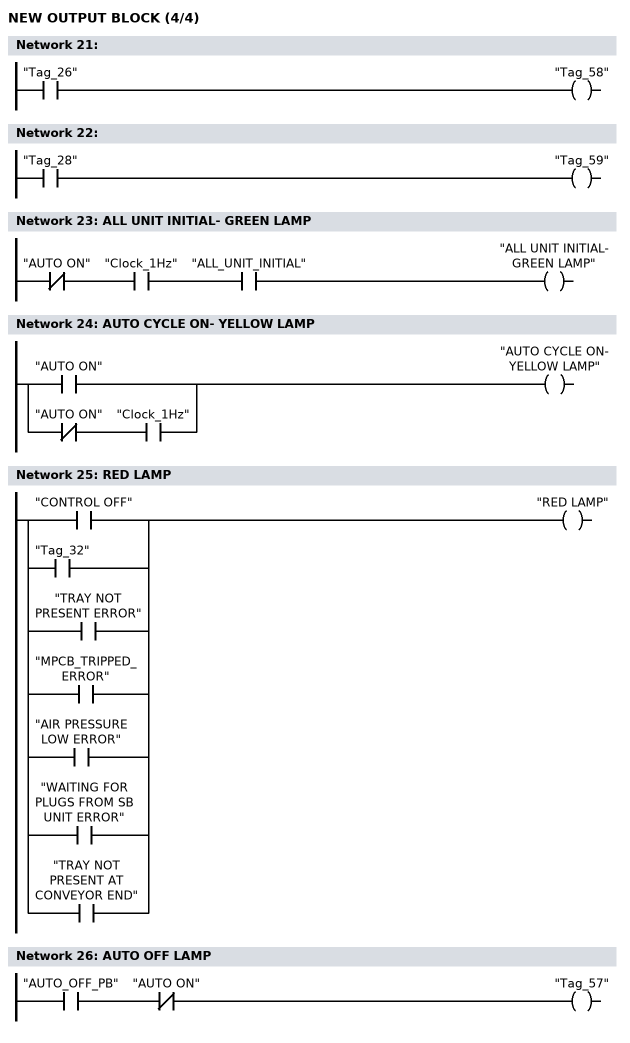
   RUNG wire#powerrail
      Contact( "Tag_26" )
      Coil( "Tag_58" )
   END_RUNG
   // the same network as SCL:
   "Tag_58" := "Tag_26";
END_REGION

REGION Network 22
   RUNG wire#powerrail
      Contact( "Tag_28" )
      Coil( "Tag_59" )
   END_RUNG
   // the same network as SCL:
   "Tag_59" := "Tag_28";
END_REGION

REGION Network 23: ALL UNIT INITIAL- GREEN LAMP
   RUNG wire#powerrail
      I_Contact( "AUTO ON" )
      Contact( "Clock_1Hz" )
      Contact( "ALL_UNIT_INITIAL" )
      Coil( "ALL UNIT INITIAL- GREEN LAMP" )
   END_RUNG
   // the same network as SCL:
   "ALL UNIT INITIAL- GREEN LAMP" := NOT "AUTO ON" AND "Clock_1Hz" AND "ALL_UNIT_INITIAL";
END_REGION

REGION Network 24: AUTO CYCLE ON- YELLOW LAMP
   RUNG wire#powerrail
      Contact( "AUTO ON" )
      wire#w1
      Coil( "AUTO CYCLE ON- YELLOW LAMP" )
   END_RUNG
   RUNG wire#powerrail
      I_Contact( "AUTO ON" )
      Contact( "Clock_1Hz" )
   END_RUNG wire#w1
   // the same network as SCL:
   "AUTO CYCLE ON- YELLOW LAMP" := "AUTO ON" OR (NOT "AUTO ON" AND "Clock_1Hz");
END_REGION

REGION Network 25: RED LAMP
   RUNG wire#powerrail
      Contact( "CONTROL OFF" )
      wire#w1
      Coil( "RED LAMP" )
   END_RUNG
   RUNG wire#powerrail
      Contact( "Tag_32" )
   END_RUNG wire#w1
   RUNG wire#powerrail
      Contact( "TRAY NOT  PRESENT ERROR" )
   END_RUNG wire#w1
   RUNG wire#powerrail
      Contact( "MPCB_TRIPPED_ERROR" )
   END_RUNG wire#w1
   RUNG wire#powerrail
      Contact( "AIR PRESSURE LOW ERROR" )
   END_RUNG wire#w1
   RUNG wire#powerrail
      Contact( "WAITING FOR PLUGS FROM SB UNIT ERROR" )
   END_RUNG wire#w1
   RUNG wire#powerrail
      Contact( "TRAY NOT PRESENT AT CONVEYOR END" )
   END_RUNG wire#w1
   // the same network as SCL:
   "RED LAMP" := "CONTROL OFF" OR "Tag_32" OR "TRAY NOT  PRESENT ERROR" OR "MPCB_TRIPPED_ERROR" OR "AIR PRESSURE LOW ERROR" OR "WAITING FOR PLUGS FROM SB UNIT ERROR" OR "TRAY NOT PRESENT AT CONVEYOR END";
END_REGION

REGION Network 26: AUTO OFF LAMP
   RUNG wire#powerrail
      Contact( "AUTO_OFF_PB" )
      I_Contact( "AUTO ON" )
      Coil( "Tag_57" )
   END_RUNG
   // the same network as SCL:
   "Tag_57" := "AUTO_OFF_PB" AND NOT "AUTO ON";
END_REGION
END_FUNCTION

FUNCTION "AUTO" : Void   // FC7, LAD
{ S7_Optimized_Access := 'TRUE' }
VERSION : 0.1
   VAR_TEMP   // added for the SCL form of the ladder/FBD networks
      _w1 : Bool;
   END_VAR
BEGIN

REGION Network 1: AUTO ON
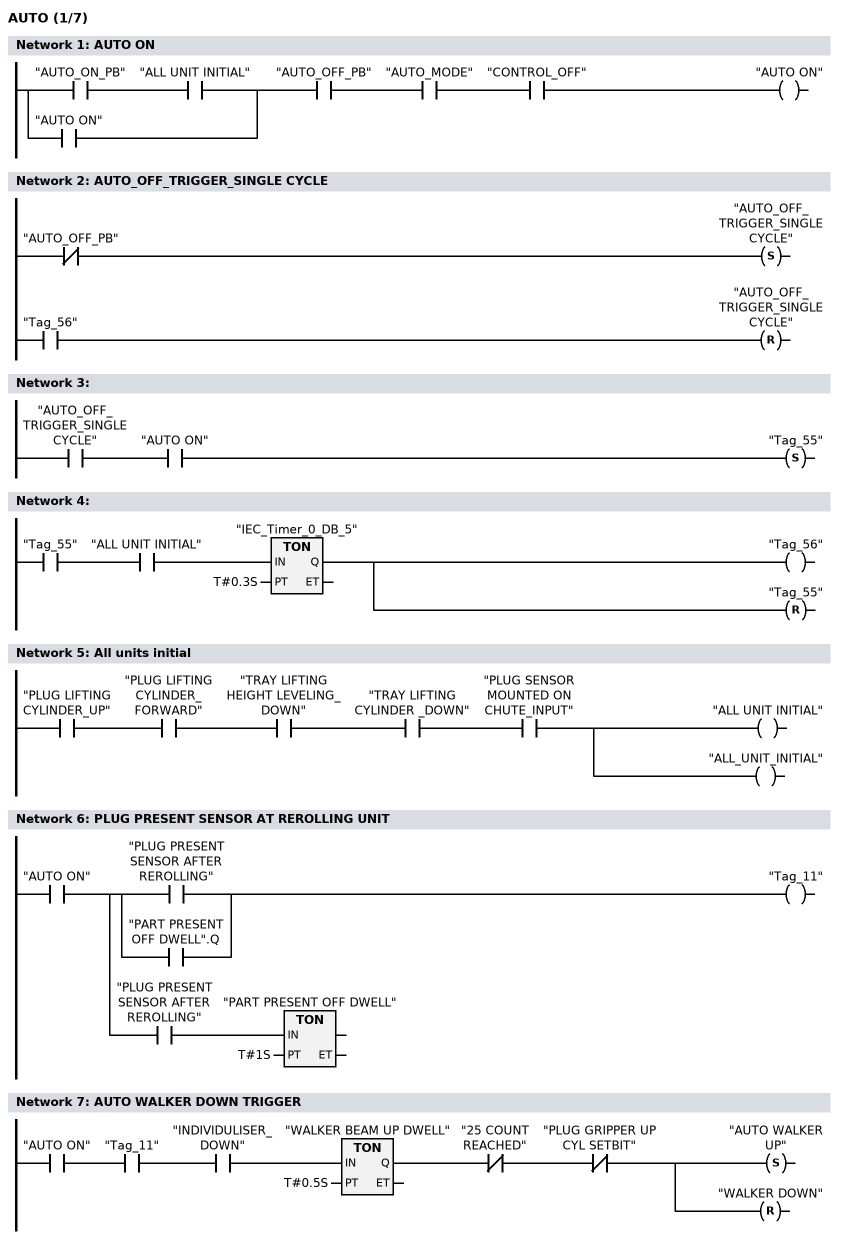
   RUNG wire#powerrail
      Contact( "AUTO_ON_PB" )
      Contact( "ALL UNIT INITIAL" )
      wire#w1
      Contact( "AUTO_OFF_PB" )
      Contact( "AUTO_MODE" )
      Contact( "CONTROL_OFF" )
      Coil( "AUTO ON" )
   END_RUNG
   RUNG wire#powerrail
      Contact( "AUTO ON" )
   END_RUNG wire#w1
   // the same network as SCL:
   "AUTO ON" := (("AUTO_ON_PB" AND "ALL UNIT INITIAL") OR "AUTO ON") AND "AUTO_OFF_PB" AND "AUTO_MODE" AND "CONTROL_OFF";
END_REGION

REGION Network 2: AUTO_OFF_TRIGGER_SINGLE CYCLE
   RUNG wire#powerrail
      I_Contact( "AUTO_OFF_PB" )
      S_Coil( "AUTO_OFF_TRIGGER_SINGLE CYCLE" )
   END_RUNG
   RUNG wire#powerrail
      Contact( "Tag_56" )
      R_Coil( "AUTO_OFF_TRIGGER_SINGLE CYCLE" )
   END_RUNG
   // the same network as SCL:
   IF NOT "AUTO_OFF_PB" THEN "AUTO_OFF_TRIGGER_SINGLE CYCLE" := TRUE; END_IF;
   IF "Tag_56" THEN "AUTO_OFF_TRIGGER_SINGLE CYCLE" := FALSE; END_IF;
END_REGION

REGION Network 3
   RUNG wire#powerrail
      Contact( "AUTO_OFF_TRIGGER_SINGLE CYCLE" )
      Contact( "AUTO ON" )
      S_Coil( "Tag_55" )
   END_RUNG
   // the same network as SCL:
   IF "AUTO_OFF_TRIGGER_SINGLE CYCLE" AND "AUTO ON" THEN "Tag_55" := TRUE; END_IF;
END_REGION

REGION Network 4
   "IEC_Timer_0_DB_5".TON(IN := "Tag_55" AND "ALL UNIT INITIAL", PT := T#0.3S);
   "Tag_56" := "IEC_Timer_0_DB_5".Q;
   IF "IEC_Timer_0_DB_5".Q THEN "Tag_55" := FALSE; END_IF;
END_REGION

REGION Network 5: All units initial
   RUNG wire#powerrail
      Contact( "PLUG LIFTING CYLINDER_UP" )
      Contact( "PLUG LIFTING CYLINDER_FORWARD" )
      Contact( "TRAY LIFTING HEIGHT LEVELING_DOWN" )
      Contact( "TRAY LIFTING CYLINDER _DOWN" )
      Contact( "PLUG SENSOR MOUNTED ON CHUTE_INPUT" )
      wire#w1
      Coil( "ALL UNIT INITIAL" )
   END_RUNG
   RUNG wire#w1
      Coil( "ALL_UNIT_INITIAL" )
   END_RUNG
   // the same network as SCL:
   "ALL UNIT INITIAL" := "PLUG LIFTING CYLINDER_UP" AND "PLUG LIFTING CYLINDER_FORWARD" AND "TRAY LIFTING HEIGHT LEVELING_DOWN" AND "TRAY LIFTING CYLINDER _DOWN" AND "PLUG SENSOR MOUNTED ON CHUTE_INPUT";
   "ALL_UNIT_INITIAL" := "ALL UNIT INITIAL";
END_REGION

REGION Network 6: PLUG PRESENT SENSOR AT REROLLING UNIT
   "Tag_11" := "AUTO ON" AND ("PLUG PRESENT SENSOR AFTER REROLLING" OR "PART PRESENT OFF DWELL".Q);
   "PART PRESENT OFF DWELL".TON(IN := "AUTO ON" AND "PLUG PRESENT SENSOR AFTER REROLLING", PT := T#1S);
END_REGION

REGION Network 7: AUTO WALKER DOWN TRIGGER
   "WALKER BEAM UP DWELL".TON(IN := "AUTO ON" AND "Tag_11" AND "INDIVIDULISER_DOWN", PT := T#0.5S);
   IF "WALKER BEAM UP DWELL".Q AND NOT "25 COUNT REACHED" AND NOT "PLUG GRIPPER UP CYL SETBIT" THEN
       "AUTO WALKER UP" := TRUE;
       "WALKER DOWN" := FALSE;
   END_IF;
END_REGION

REGION Network 8
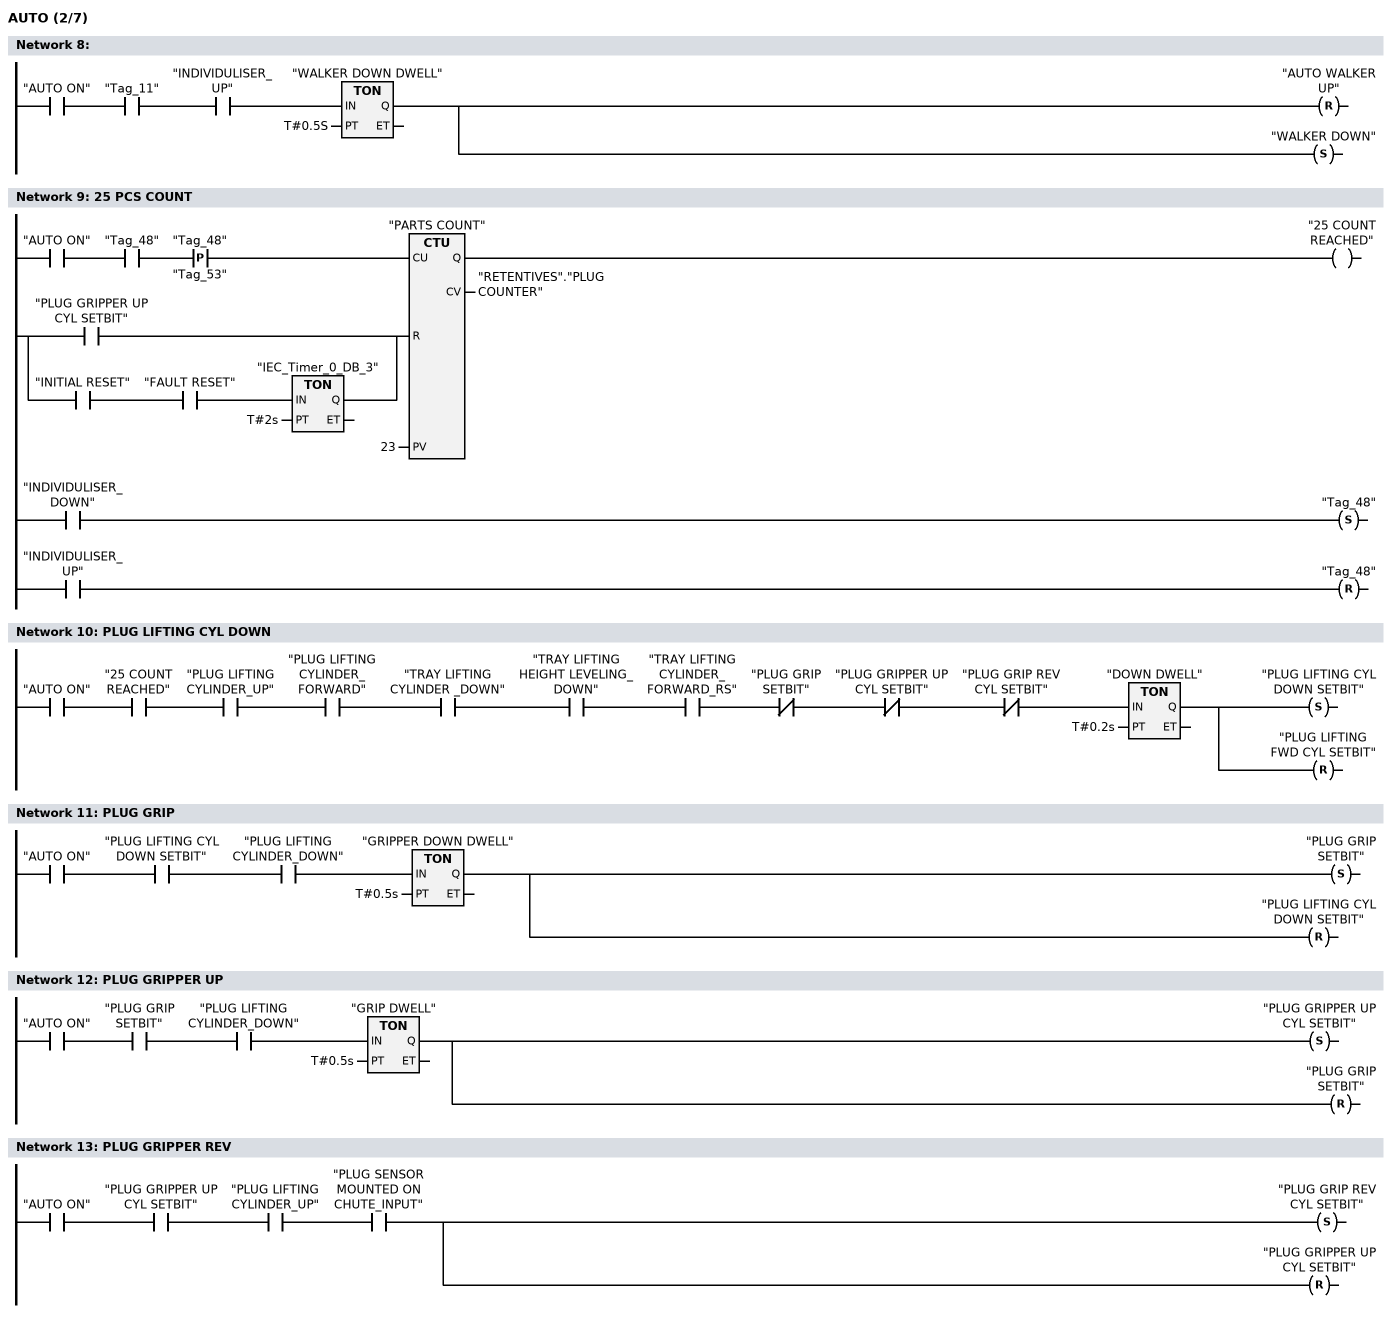
   "WALKER DOWN DWELL".TON(IN := "AUTO ON" AND "Tag_11" AND "INDIVIDULISER_UP", PT := T#0.5S);
   IF "WALKER DOWN DWELL".Q THEN
       "AUTO WALKER UP" := FALSE;
       "WALKER DOWN" := TRUE;
   END_IF;
END_REGION

REGION Network 9: 25 PCS COUNT
   #_w1 := "AUTO ON" AND "Tag_48" AND "Tag_48" AND NOT "Tag_53";   // rising edge of "Tag_48"
   "Tag_53" := "Tag_48";
   "IEC_Timer_0_DB_3".TON(IN := "INITIAL RESET" AND "FAULT RESET", PT := T#2s);
   "PARTS COUNT".CTU(CU := #_w1,
                     R := "PLUG GRIPPER UP CYL SETBIT" OR "IEC_Timer_0_DB_3".Q,
                     PV := 23,
                     CV => "RETENTIVES"."PLUG COUNTER");
   "25 COUNT REACHED" := "PARTS COUNT".Q;
   IF "INDIVIDULISER_DOWN" THEN "Tag_48" := TRUE; END_IF;
   IF "INDIVIDULISER_UP" THEN "Tag_48" := FALSE; END_IF;
END_REGION

REGION Network 10: PLUG LIFTING CYL DOWN
   "DOWN DWELL".TON(IN := "AUTO ON" AND "25 COUNT REACHED" AND "PLUG LIFTING CYLINDER_UP" AND "PLUG LIFTING CYLINDER_FORWARD" AND "TRAY LIFTING CYLINDER _DOWN" AND "TRAY LIFTING HEIGHT LEVELING_DOWN" AND "TRAY LIFTING CYLINDER_FORWARD_RS" AND NOT "PLUG GRIP SETBIT" AND NOT "PLUG GRIPPER UP CYL SETBIT" AND NOT "PLUG GRIP REV CYL SETBIT",
                    PT := T#0.2s);
   IF "DOWN DWELL".Q THEN
       "PLUG LIFTING CYL DOWN SETBIT" := TRUE;
       "PLUG LIFTING FWD CYL SETBIT" := FALSE;
   END_IF;
END_REGION

REGION Network 11: PLUG GRIP
   "GRIPPER DOWN DWELL".TON(IN := "AUTO ON" AND "PLUG LIFTING CYL DOWN SETBIT" AND "PLUG LIFTING CYLINDER_DOWN",
                           PT := T#0.5s);
   IF "GRIPPER DOWN DWELL".Q THEN
       "PLUG GRIP SETBIT" := TRUE;
       "PLUG LIFTING CYL DOWN SETBIT" := FALSE;
   END_IF;
END_REGION

REGION Network 12: PLUG GRIPPER UP
   "GRIP DWELL".TON(IN := "AUTO ON" AND "PLUG GRIP SETBIT" AND "PLUG LIFTING CYLINDER_DOWN", PT := T#0.5s);
   IF "GRIP DWELL".Q THEN
       "PLUG GRIPPER UP CYL SETBIT" := TRUE;
       "PLUG GRIP SETBIT" := FALSE;
   END_IF;
END_REGION

REGION Network 13: PLUG GRIPPER REV
   RUNG wire#powerrail
      Contact( "AUTO ON" )
      Contact( "PLUG GRIPPER UP CYL SETBIT" )
      Contact( "PLUG LIFTING CYLINDER_UP" )
      Contact( "PLUG SENSOR MOUNTED ON CHUTE_INPUT" )
      wire#w1
      S_Coil( "PLUG GRIP REV CYL SETBIT" )
   END_RUNG
   RUNG wire#w1
      R_Coil( "PLUG GRIPPER UP CYL SETBIT" )
   END_RUNG
   // the same network as SCL:
   IF "AUTO ON" AND "PLUG GRIPPER UP CYL SETBIT" AND "PLUG LIFTING CYLINDER_UP" AND "PLUG SENSOR MOUNTED ON CHUTE_INPUT" THEN
       "PLUG GRIP REV CYL SETBIT" := TRUE;
       "PLUG GRIPPER UP CYL SETBIT" := FALSE;
   END_IF;
END_REGION

REGION Network 14: PLUG LIFTING CYL DOWN AT TRAY
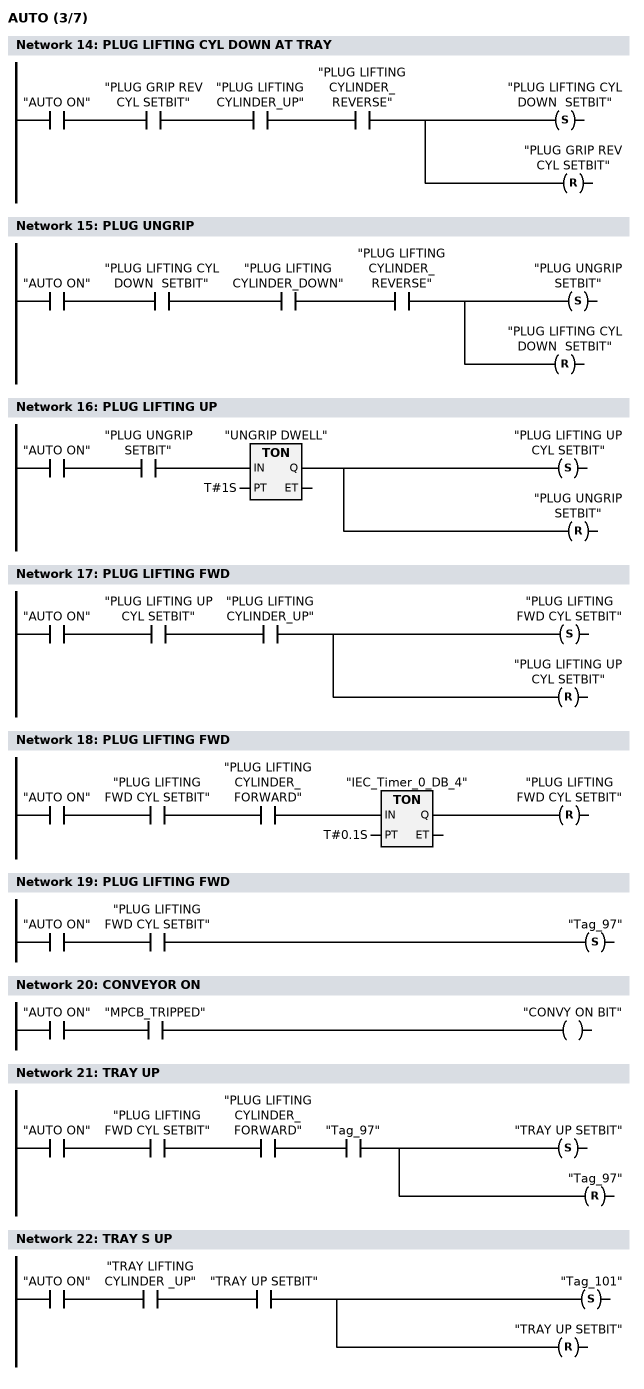
   RUNG wire#powerrail
      Contact( "AUTO ON" )
      Contact( "PLUG GRIP REV CYL SETBIT" )
      Contact( "PLUG LIFTING CYLINDER_UP" )
      Contact( "PLUG LIFTING CYLINDER_REVERSE" )
      wire#w1
      S_Coil( "PLUG LIFTING CYL DOWN  SETBIT" )
   END_RUNG
   RUNG wire#w1
      R_Coil( "PLUG GRIP REV CYL SETBIT" )
   END_RUNG
   // the same network as SCL:
   IF "AUTO ON" AND "PLUG GRIP REV CYL SETBIT" AND "PLUG LIFTING CYLINDER_UP" AND "PLUG LIFTING CYLINDER_REVERSE" THEN
       "PLUG LIFTING CYL DOWN  SETBIT" := TRUE;
       "PLUG GRIP REV CYL SETBIT" := FALSE;
   END_IF;
END_REGION

REGION Network 15: PLUG UNGRIP
   RUNG wire#powerrail
      Contact( "AUTO ON" )
      Contact( "PLUG LIFTING CYL DOWN  SETBIT" )
      Contact( "PLUG LIFTING CYLINDER_DOWN" )
      Contact( "PLUG LIFTING CYLINDER_REVERSE" )
      wire#w1
      S_Coil( "PLUG UNGRIP SETBIT" )
   END_RUNG
   RUNG wire#w1
      R_Coil( "PLUG LIFTING CYL DOWN  SETBIT" )
   END_RUNG
   // the same network as SCL:
   IF "AUTO ON" AND "PLUG LIFTING CYL DOWN  SETBIT" AND "PLUG LIFTING CYLINDER_DOWN" AND "PLUG LIFTING CYLINDER_REVERSE" THEN
       "PLUG UNGRIP SETBIT" := TRUE;
       "PLUG LIFTING CYL DOWN  SETBIT" := FALSE;
   END_IF;
END_REGION

REGION Network 16: PLUG LIFTING UP
   "UNGRIP DWELL".TON(IN := "AUTO ON" AND "PLUG UNGRIP SETBIT", PT := T#1S);
   IF "UNGRIP DWELL".Q THEN
       "PLUG LIFTING UP CYL SETBIT" := TRUE;
       "PLUG UNGRIP SETBIT" := FALSE;
   END_IF;
END_REGION

REGION Network 17: PLUG LIFTING FWD
   RUNG wire#powerrail
      Contact( "AUTO ON" )
      Contact( "PLUG LIFTING UP CYL SETBIT" )
      Contact( "PLUG LIFTING CYLINDER_UP" )
      wire#w1
      S_Coil( "PLUG LIFTING FWD CYL SETBIT" )
   END_RUNG
   RUNG wire#w1
      R_Coil( "PLUG LIFTING UP CYL SETBIT" )
   END_RUNG
   // the same network as SCL:
   IF "AUTO ON" AND "PLUG LIFTING UP CYL SETBIT" AND "PLUG LIFTING CYLINDER_UP" THEN
       "PLUG LIFTING FWD CYL SETBIT" := TRUE;
       "PLUG LIFTING UP CYL SETBIT" := FALSE;
   END_IF;
END_REGION

REGION Network 18: PLUG LIFTING FWD
   "IEC_Timer_0_DB_4".TON(IN := "AUTO ON" AND "PLUG LIFTING FWD CYL SETBIT" AND "PLUG LIFTING CYLINDER_FORWARD",
                          PT := T#0.1S);
   IF "IEC_Timer_0_DB_4".Q THEN "PLUG LIFTING FWD CYL SETBIT" := FALSE; END_IF;
END_REGION

REGION Network 19: PLUG LIFTING FWD
   RUNG wire#powerrail
      Contact( "AUTO ON" )
      Contact( "PLUG LIFTING FWD CYL SETBIT" )
      S_Coil( "Tag_97" )
   END_RUNG
   // the same network as SCL:
   IF "AUTO ON" AND "PLUG LIFTING FWD CYL SETBIT" THEN "Tag_97" := TRUE; END_IF;
END_REGION

REGION Network 20: CONVEYOR ON
   RUNG wire#powerrail
      Contact( "AUTO ON" )
      Contact( "MPCB_TRIPPED" )
      Coil( "CONVY ON BIT" )
   END_RUNG
   // the same network as SCL:
   "CONVY ON BIT" := "AUTO ON" AND "MPCB_TRIPPED";
END_REGION

REGION Network 21: TRAY UP
   RUNG wire#powerrail
      Contact( "AUTO ON" )
      Contact( "PLUG LIFTING FWD CYL SETBIT" )
      Contact( "PLUG LIFTING CYLINDER_FORWARD" )
      Contact( "Tag_97" )
      wire#w1
      S_Coil( "TRAY UP SETBIT" )
   END_RUNG
   RUNG wire#w1
      R_Coil( "Tag_97" )
   END_RUNG
   // the same network as SCL:
   IF "AUTO ON" AND "PLUG LIFTING FWD CYL SETBIT" AND "PLUG LIFTING CYLINDER_FORWARD" AND "Tag_97" THEN
       "TRAY UP SETBIT" := TRUE;
       "Tag_97" := FALSE;
   END_IF;
END_REGION

REGION Network 22: TRAY S UP
   RUNG wire#powerrail
      Contact( "AUTO ON" )
      Contact( "TRAY LIFTING CYLINDER _UP" )
      Contact( "TRAY UP SETBIT" )
      wire#w1
      S_Coil( "Tag_101" )
   END_RUNG
   RUNG wire#w1
      R_Coil( "TRAY UP SETBIT" )
   END_RUNG
   // the same network as SCL:
   IF "AUTO ON" AND "TRAY LIFTING CYLINDER _UP" AND "TRAY UP SETBIT" THEN
       "Tag_101" := TRUE;
       "TRAY UP SETBIT" := FALSE;
   END_IF;
END_REGION

REGION Network 23: TRAY REV
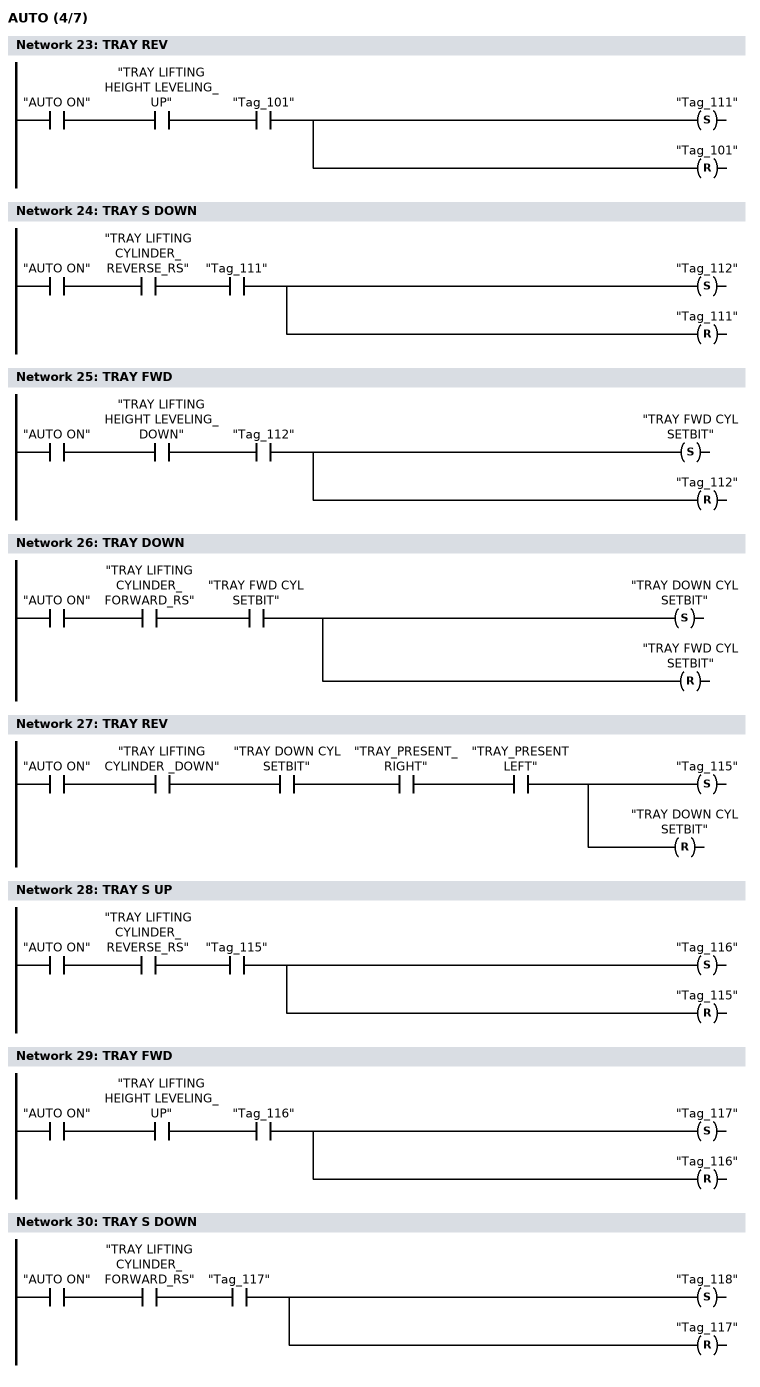
   RUNG wire#powerrail
      Contact( "AUTO ON" )
      Contact( "TRAY LIFTING HEIGHT LEVELING_UP" )
      Contact( "Tag_101" )
      wire#w1
      S_Coil( "Tag_111" )
   END_RUNG
   RUNG wire#w1
      R_Coil( "Tag_101" )
   END_RUNG
   // the same network as SCL:
   IF "AUTO ON" AND "TRAY LIFTING HEIGHT LEVELING_UP" AND "Tag_101" THEN
       "Tag_111" := TRUE;
       "Tag_101" := FALSE;
   END_IF;
END_REGION

REGION Network 24: TRAY S DOWN
   RUNG wire#powerrail
      Contact( "AUTO ON" )
      Contact( "TRAY LIFTING CYLINDER_REVERSE_RS" )
      Contact( "Tag_111" )
      wire#w1
      S_Coil( "Tag_112" )
   END_RUNG
   RUNG wire#w1
      R_Coil( "Tag_111" )
   END_RUNG
   // the same network as SCL:
   IF "AUTO ON" AND "TRAY LIFTING CYLINDER_REVERSE_RS" AND "Tag_111" THEN
       "Tag_112" := TRUE;
       "Tag_111" := FALSE;
   END_IF;
END_REGION

REGION Network 25: TRAY FWD
   RUNG wire#powerrail
      Contact( "AUTO ON" )
      Contact( "TRAY LIFTING HEIGHT LEVELING_DOWN" )
      Contact( "Tag_112" )
      wire#w1
      S_Coil( "TRAY FWD CYL SETBIT" )
   END_RUNG
   RUNG wire#w1
      R_Coil( "Tag_112" )
   END_RUNG
   // the same network as SCL:
   IF "AUTO ON" AND "TRAY LIFTING HEIGHT LEVELING_DOWN" AND "Tag_112" THEN
       "TRAY FWD CYL SETBIT" := TRUE;
       "Tag_112" := FALSE;
   END_IF;
END_REGION

REGION Network 26: TRAY DOWN
   RUNG wire#powerrail
      Contact( "AUTO ON" )
      Contact( "TRAY LIFTING CYLINDER_FORWARD_RS" )
      Contact( "TRAY FWD CYL SETBIT" )
      wire#w1
      S_Coil( "TRAY DOWN CYL SETBIT" )
   END_RUNG
   RUNG wire#w1
      R_Coil( "TRAY FWD CYL SETBIT" )
   END_RUNG
   // the same network as SCL:
   IF "AUTO ON" AND "TRAY LIFTING CYLINDER_FORWARD_RS" AND "TRAY FWD CYL SETBIT" THEN
       "TRAY DOWN CYL SETBIT" := TRUE;
       "TRAY FWD CYL SETBIT" := FALSE;
   END_IF;
END_REGION

REGION Network 27: TRAY REV
   RUNG wire#powerrail
      Contact( "AUTO ON" )
      Contact( "TRAY LIFTING CYLINDER _DOWN" )
      Contact( "TRAY DOWN CYL SETBIT" )
      Contact( "TRAY_PRESENT_RIGHT" )
      Contact( "TRAY_PRESENT LEFT" )
      wire#w1
      S_Coil( "Tag_115" )
   END_RUNG
   RUNG wire#w1
      R_Coil( "TRAY DOWN CYL SETBIT" )
   END_RUNG
   // the same network as SCL:
   IF "AUTO ON" AND "TRAY LIFTING CYLINDER _DOWN" AND "TRAY DOWN CYL SETBIT" AND "TRAY_PRESENT_RIGHT" AND "TRAY_PRESENT LEFT" THEN
       "Tag_115" := TRUE;
       "TRAY DOWN CYL SETBIT" := FALSE;
   END_IF;
END_REGION

REGION Network 28: TRAY S UP
   RUNG wire#powerrail
      Contact( "AUTO ON" )
      Contact( "TRAY LIFTING CYLINDER_REVERSE_RS" )
      Contact( "Tag_115" )
      wire#w1
      S_Coil( "Tag_116" )
   END_RUNG
   RUNG wire#w1
      R_Coil( "Tag_115" )
   END_RUNG
   // the same network as SCL:
   IF "AUTO ON" AND "TRAY LIFTING CYLINDER_REVERSE_RS" AND "Tag_115" THEN
       "Tag_116" := TRUE;
       "Tag_115" := FALSE;
   END_IF;
END_REGION

REGION Network 29: TRAY FWD
   RUNG wire#powerrail
      Contact( "AUTO ON" )
      Contact( "TRAY LIFTING HEIGHT LEVELING_UP" )
      Contact( "Tag_116" )
      wire#w1
      S_Coil( "Tag_117" )
   END_RUNG
   RUNG wire#w1
      R_Coil( "Tag_116" )
   END_RUNG
   // the same network as SCL:
   IF "AUTO ON" AND "TRAY LIFTING HEIGHT LEVELING_UP" AND "Tag_116" THEN
       "Tag_117" := TRUE;
       "Tag_116" := FALSE;
   END_IF;
END_REGION

REGION Network 30: TRAY S DOWN
   RUNG wire#powerrail
      Contact( "AUTO ON" )
      Contact( "TRAY LIFTING CYLINDER_FORWARD_RS" )
      Contact( "Tag_117" )
      wire#w1
      S_Coil( "Tag_118" )
   END_RUNG
   RUNG wire#w1
      R_Coil( "Tag_117" )
   END_RUNG
   // the same network as SCL:
   IF "AUTO ON" AND "TRAY LIFTING CYLINDER_FORWARD_RS" AND "Tag_117" THEN
       "Tag_118" := TRUE;
       "Tag_117" := FALSE;
   END_IF;
END_REGION

REGION Network 31: TRAY S DOWN
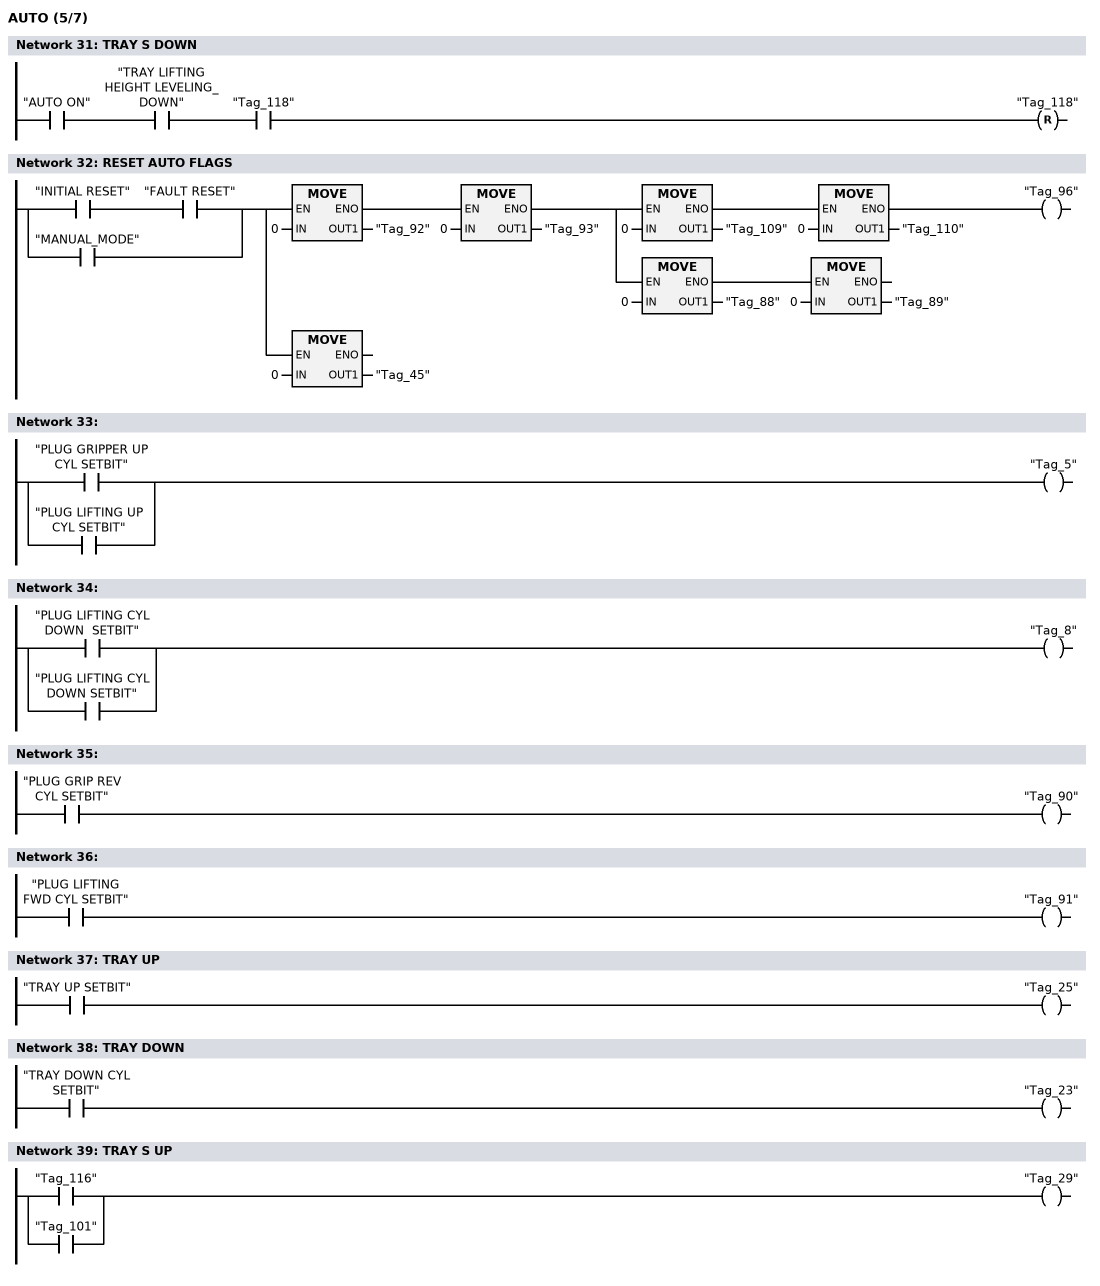
   RUNG wire#powerrail
      Contact( "AUTO ON" )
      Contact( "TRAY LIFTING HEIGHT LEVELING_DOWN" )
      Contact( "Tag_118" )
      R_Coil( "Tag_118" )
   END_RUNG
   // the same network as SCL:
   IF "AUTO ON" AND "TRAY LIFTING HEIGHT LEVELING_DOWN" AND "Tag_118" THEN "Tag_118" := FALSE; END_IF;
END_REGION

REGION Network 32: RESET AUTO FLAGS
   RUNG wire#powerrail
      Contact( "INITIAL RESET" )
      Contact( "FAULT RESET" )
      wire#w1
      Move(in := 0, out1 => "Tag_92")
      Move(in := 0, out1 => "Tag_93")
      wire#w2
      Move(in := 0, out1 => "Tag_109")
      Move(in := 0, out1 => "Tag_110")
      Coil( "Tag_96" )
   END_RUNG
   RUNG wire#powerrail
      Contact( "MANUAL_MODE" )
   END_RUNG wire#w1
   RUNG wire#w2
      Move(in := 0, out1 => "Tag_88")
      Move(in := 0, out1 => "Tag_89")
   END_RUNG
   RUNG wire#w1
      Move(in := 0, out1 => "Tag_45")
   END_RUNG
   // the same network as SCL:
   #_w1 := ("INITIAL RESET" AND "FAULT RESET") OR "MANUAL_MODE";
   IF #_w1 THEN
       "Tag_92" := 0;
       "Tag_93" := 0;
       "Tag_109" := 0;
       "Tag_110" := 0;
   END_IF;
   "Tag_96" := #_w1;
   IF #_w1 THEN
       "Tag_88" := 0;
       "Tag_89" := 0;
       "Tag_45" := 0;
   END_IF;
END_REGION

REGION Network 33
   RUNG wire#powerrail
      Contact( "PLUG GRIPPER UP CYL SETBIT" )
      wire#w1
      Coil( "Tag_5" )
   END_RUNG
   RUNG wire#powerrail
      Contact( "PLUG LIFTING UP CYL SETBIT" )
   END_RUNG wire#w1
   // the same network as SCL:
   "Tag_5" := "PLUG GRIPPER UP CYL SETBIT" OR "PLUG LIFTING UP CYL SETBIT";
END_REGION

REGION Network 34
   RUNG wire#powerrail
      Contact( "PLUG LIFTING CYL DOWN  SETBIT" )
      wire#w1
      Coil( "Tag_8" )
   END_RUNG
   RUNG wire#powerrail
      Contact( "PLUG LIFTING CYL DOWN SETBIT" )
   END_RUNG wire#w1
   // the same network as SCL:
   "Tag_8" := "PLUG LIFTING CYL DOWN  SETBIT" OR "PLUG LIFTING CYL DOWN SETBIT";
END_REGION

REGION Network 35
   RUNG wire#powerrail
      Contact( "PLUG GRIP REV CYL SETBIT" )
      Coil( "Tag_90" )
   END_RUNG
   // the same network as SCL:
   "Tag_90" := "PLUG GRIP REV CYL SETBIT";
END_REGION

REGION Network 36
   RUNG wire#powerrail
      Contact( "PLUG LIFTING FWD CYL SETBIT" )
      Coil( "Tag_91" )
   END_RUNG
   // the same network as SCL:
   "Tag_91" := "PLUG LIFTING FWD CYL SETBIT";
END_REGION

REGION Network 37: TRAY UP
   RUNG wire#powerrail
      Contact( "TRAY UP SETBIT" )
      Coil( "Tag_25" )
   END_RUNG
   // the same network as SCL:
   "Tag_25" := "TRAY UP SETBIT";
END_REGION

REGION Network 38: TRAY DOWN
   RUNG wire#powerrail
      Contact( "TRAY DOWN CYL SETBIT" )
      Coil( "Tag_23" )
   END_RUNG
   // the same network as SCL:
   "Tag_23" := "TRAY DOWN CYL SETBIT";
END_REGION

REGION Network 39: TRAY S UP
   RUNG wire#powerrail
      Contact( "Tag_116" )
      wire#w1
      Coil( "Tag_29" )
   END_RUNG
   RUNG wire#powerrail
      Contact( "Tag_101" )
   END_RUNG wire#w1
   // the same network as SCL:
   "Tag_29" := "Tag_116" OR "Tag_101";
END_REGION

REGION Network 40: TRAY S DOWN
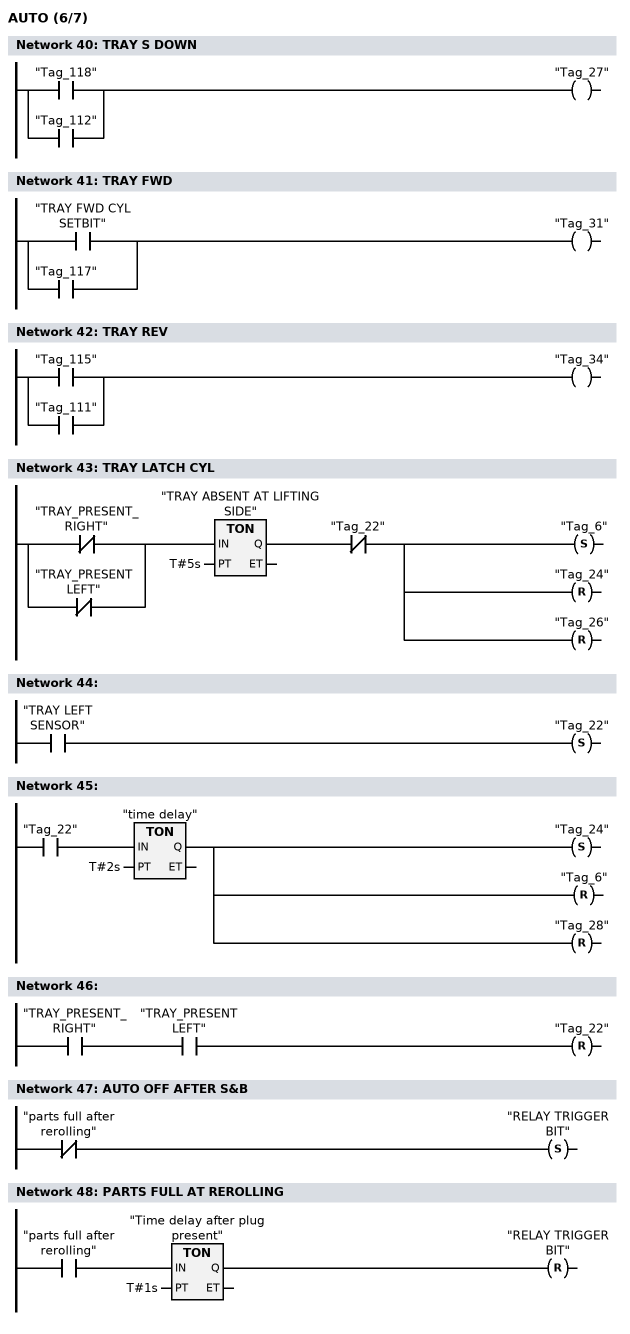
   RUNG wire#powerrail
      Contact( "Tag_118" )
      wire#w1
      Coil( "Tag_27" )
   END_RUNG
   RUNG wire#powerrail
      Contact( "Tag_112" )
   END_RUNG wire#w1
   // the same network as SCL:
   "Tag_27" := "Tag_118" OR "Tag_112";
END_REGION

REGION Network 41: TRAY FWD
   RUNG wire#powerrail
      Contact( "TRAY FWD CYL SETBIT" )
      wire#w1
      Coil( "Tag_31" )
   END_RUNG
   RUNG wire#powerrail
      Contact( "Tag_117" )
   END_RUNG wire#w1
   // the same network as SCL:
   "Tag_31" := "TRAY FWD CYL SETBIT" OR "Tag_117";
END_REGION

REGION Network 42: TRAY REV
   RUNG wire#powerrail
      Contact( "Tag_115" )
      wire#w1
      Coil( "Tag_34" )
   END_RUNG
   RUNG wire#powerrail
      Contact( "Tag_111" )
   END_RUNG wire#w1
   // the same network as SCL:
   "Tag_34" := "Tag_115" OR "Tag_111";
END_REGION

REGION Network 43: TRAY LATCH CYL
   "TRAY ABSENT AT LIFTING SIDE".TON(IN := NOT "TRAY_PRESENT_RIGHT" OR NOT "TRAY_PRESENT LEFT", PT := T#5s);
   IF "TRAY ABSENT AT LIFTING SIDE".Q AND NOT "Tag_22" THEN
       "Tag_6" := TRUE;
       "Tag_24" := FALSE;
       "Tag_26" := FALSE;
   END_IF;
END_REGION

REGION Network 44
   RUNG wire#powerrail
      Contact( "TRAY LEFT SENSOR" )
      S_Coil( "Tag_22" )
   END_RUNG
   // the same network as SCL:
   IF "TRAY LEFT SENSOR" THEN "Tag_22" := TRUE; END_IF;
END_REGION

REGION Network 45
   "time delay".TON(IN := "Tag_22", PT := T#2s);
   IF "time delay".Q THEN
       "Tag_24" := TRUE;
       "Tag_6" := FALSE;
       "Tag_28" := FALSE;
   END_IF;
END_REGION

REGION Network 46
   RUNG wire#powerrail
      Contact( "TRAY_PRESENT_RIGHT" )
      Contact( "TRAY_PRESENT LEFT" )
      R_Coil( "Tag_22" )
   END_RUNG
   // the same network as SCL:
   IF "TRAY_PRESENT_RIGHT" AND "TRAY_PRESENT LEFT" THEN "Tag_22" := FALSE; END_IF;
END_REGION

REGION Network 47: AUTO OFF AFTER S&B
   RUNG wire#powerrail
      I_Contact( "parts full after rerolling" )
      S_Coil( "RELAY TRIGGER BIT" )
   END_RUNG
   // the same network as SCL:
   IF NOT "parts full after rerolling" THEN "RELAY TRIGGER BIT" := TRUE; END_IF;
END_REGION

REGION Network 48: PARTS FULL AT REROLLING
   "Time delay after plug present".TON(IN := "parts full after rerolling", PT := T#1s);
   IF "Time delay after plug present".Q THEN "RELAY TRIGGER BIT" := FALSE; END_IF;
END_REGION

REGION Network 49: TRAY STOPPER UP
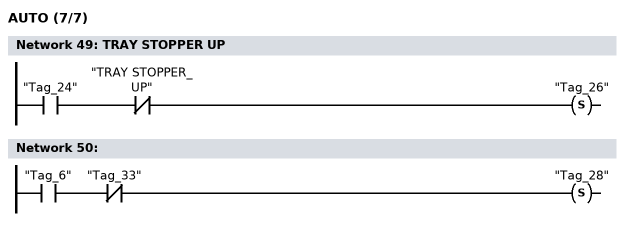
   RUNG wire#powerrail
      Contact( "Tag_24" )
      I_Contact( "TRAY STOPPER_UP" )
      S_Coil( "Tag_26" )
   END_RUNG
   // the same network as SCL:
   IF "Tag_24" AND NOT "TRAY STOPPER_UP" THEN "Tag_26" := TRUE; END_IF;
END_REGION

REGION Network 50
   RUNG wire#powerrail
      Contact( "Tag_6" )
      I_Contact( "Tag_33" )
      S_Coil( "Tag_28" )
   END_RUNG
   // the same network as SCL:
   IF "Tag_6" AND NOT "Tag_33" THEN "Tag_28" := TRUE; END_IF;
END_REGION
END_FUNCTION

ORGANIZATION_BLOCK "Main"   // OB1, LAD, ProgramCycle
TITLE = "Main Program Sweep (Cycle)"
{ S7_Optimized_Access := 'TRUE' }
VERSION : 0.1
   VAR_INPUT
      Initial_Call : Bool;   // Initial call of this OB
      Remanence : Bool;   // =True, if remanent data are available
   END_VAR
   VAR_TEMP   // added for the SCL form of the ladder/FBD networks
      _w1 : Bool;
   END_VAR
BEGIN

REGION Network 1
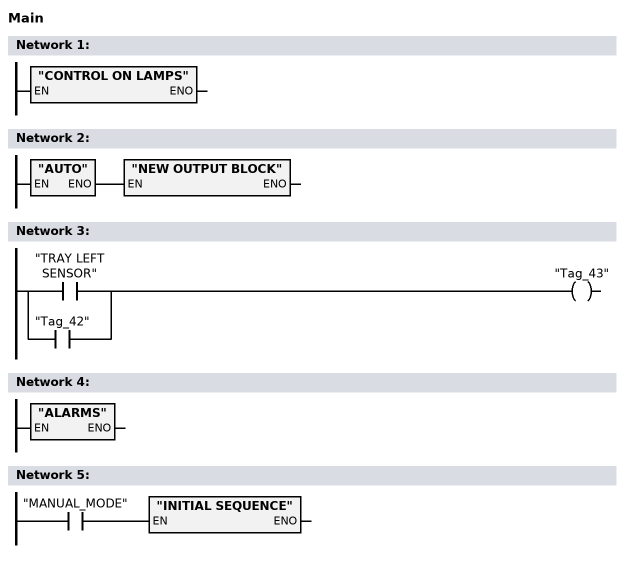
   RUNG wire#powerrail
      "CONTROL ON LAMPS"()
   END_RUNG
   // the same network as SCL:
   "CONTROL ON LAMPS"();
END_REGION

REGION Network 2
   RUNG wire#powerrail
      "AUTO"()
      "NEW OUTPUT BLOCK"()
   END_RUNG
   // the same network as SCL:
   "AUTO"(ENO => #_w1);
   IF #_w1 THEN "NEW OUTPUT BLOCK"(); END_IF;
END_REGION

REGION Network 3
   RUNG wire#powerrail
      Contact( "TRAY LEFT SENSOR" )
      wire#w1
      Coil( "Tag_43" )
   END_RUNG
   RUNG wire#powerrail
      Contact( "Tag_42" )
   END_RUNG wire#w1
   // the same network as SCL:
   "Tag_43" := "TRAY LEFT SENSOR" OR "Tag_42";
END_REGION

REGION Network 4
   RUNG wire#powerrail
      "ALARMS"()
   END_RUNG
   // the same network as SCL:
   "ALARMS"();
END_REGION

REGION Network 5
   RUNG wire#powerrail
      Contact( "MANUAL_MODE" )
      "INITIAL SEQUENCE"()
   END_RUNG
   // the same network as SCL:
   IF "MANUAL_MODE" THEN "INITIAL SEQUENCE"(); END_IF;
END_REGION
END_ORGANIZATION_BLOCK

(* ===== HMI "HMI_RT_1" =====
system functions are stored by id; their names below are inferred from use
connection "HMI_Connection_1": ETHERNET, SMART_S7_1200_OMS

HMI tags "Default tag table"
   "System_Byte" : Byte = PLC System_Byte AT %MB1, 1 s
   "RETENTIVES_PLUG COUNTER" : DInt = PLC RETENTIVES."PLUG COUNTER" AT %DB3.DBD0, 100 ms
   "Clock_Byte" : Byte = PLC Clock_Byte AT %MB0, 1 s
   "INDIVIDUAL CYLINDER UP FROM HMI" : Bool = PLC "INDIVIDUAL CYLINDER UP FROM HMI" AT %M104.5, 1 s
   "INDIVIDUAL CYLINDER DOWN FROM HMI" : Bool = PLC "INDIVIDUAL CYLINDER DOWN FROM HMI" AT %M104.6, 1 s
   "TRAY LIFTING HEIGHT LEVELING UP FROM HMI" : Bool = PLC "TRAY LIFTING HEIGHT LEVELING UP FROM HMI" AT %M104.7, 1 s
   "TRAY LIFTING HEIGHT LEVELING DOWN FROM HMI" : Bool = PLC "TRAY LIFTING HEIGHT LEVELING DOWN FROM HMI" AT %M105.0, 1 s
   "TRAY LIFTING CYLINDER  UP FROM HMI" : Bool = PLC "TRAY LIFTING CYLINDER  UP FROM HMI" AT %M105.1, 1 s
   "TRAY LIFTING CYLINDER  DOWN FROM HMI" : Bool = PLC "TRAY LIFTING CYLINDER  DOWN FROM HMI" AT %M105.2, 1 s
   "TRAY LIFTING CYLINDER FORWARD FROM HMI" : Bool = PLC "TRAY LIFTING CYLINDER FORWARD FROM HMI" AT %M105.3, 1 s
   "TRAY LIFTING CYLINDER REVERSE FROM HMI" : Bool = PLC "TRAY LIFTING CYLINDER REVERSE FROM HMI" AT %M105.4, 1 s
   "PLUG LIFTING CYLINDER UP FROM HMI" : Bool = PLC "PLUG LIFTING CYLINDER UP FROM HMI" AT %M105.5, 1 s
   "PLUG LIFTING CYLINDER REVERSE FROM HMI" : Bool = PLC "PLUG LIFTING CYLINDER REVERSE FROM HMI" AT %M106.0, 1 s
   "PLUG LIFTING CYLINDER FORWARD FROM HMI" : Bool = PLC "PLUG LIFTING CYLINDER FORWARD FROM HMI" AT %M105.7, 1 s
   "TRAY STOPPER UP FROM HMI" : Bool = PLC "TRAY STOPPER UP FROM HMI" AT %M106.1, 1 s
   "TRAY STOPPER DOWN FROM HMI" : Bool = PLC "TRAY STOPPER DOWN FROM HMI" AT %M106.2, 1 s
   "TRAY LATCH UP FROM HMI" : Bool = PLC "TRAY LATCH UP FROM HMI" AT %M106.3, 1 s
   "TRAY LATCH DOWN FROM HMI" : Bool = PLC "TRAY LATCH DOWN FROM HMI" AT %M106.4, 1 s
   "CONVEYOR -1 RUN FROM HMI" : Bool = PLC "CONVEYOR -1 RUN FROM HMI" AT %M100.0, 1 s
   "CONVEYOR -1 STOP FROM HMI" : Bool = PLC "CONVEYOR -1 STOP FROM HMI" AT %M107.1, 1 s
   "CONVEYOR 2 RUN FROM HMI" : Bool = PLC "CONVEYOR 2 RUN FROM HMI" AT %M100.1, 1 s
   "CONVEYOR -2 STOP FROM HMI" : Bool = PLC "CONVEYOR -2 STOP FROM HMI" AT %M107.2, 1 s
   "PLUG LIFTING CYLINDER  DOWN FROM HMI" : Bool = PLC "PLUG LIFTING CYLINDER  DOWN FROM HMI" AT %M105.6, 1 s
   "PLUG HOLD FROM HMI" : Bool = PLC "PLUG HOLD FROM HMI" AT %M107.3, 1 s
   "PLUD UNHOLD FROM HMI" : Bool = PLC "PLUD UNHOLD FROM HMI" AT %M107.4, 1 s
   "RETENTIVES_ERROR MSGS MOV BIT" : DInt = PLC RETENTIVES."ERROR MSGS MOV BIT" AT %DB3.DBD12, 1 s
   "down tray present by pass on" : Bool = PLC "down tray present by pass on" AT %M25.5, 1 s
   "Tag_27" : Bool = PLC "TRAY LIFTING CYLINDER_REVERSE_RS" AT %I3.2, 1 s
   "Tag_31" : Bool = PLC "PLUG LIFTING CYLINDER_REVERSE" AT %I3.6, 1 s
   "Tag_23" : Bool = PLC "TRAY LIFTING HEIGHT LEVELING_DOWN" AT %I2.6, 1 s
   "Tag_25" : Bool = PLC "TRAY LIFTING CYLINDER _DOWN" AT %I3.0, 1 s
   "Tag_28" : Bool = PLC "PLUG LIFTING CYLINDER_UP" AT %I3.4, 1 s
   "Tag_11" : Bool = PLC "WALKER BEAM DOWN" AT %Q0.1, 1 s
   "Tag_12" : Bool = PLC Tag_12 AT %Q1.0, 1 s
   "Tag_13" : Bool = PLC Tag_13 AT %Q1.1, 1 s
   "Tag_48" : Bool = PLC GRIPPER_HOLD AT %Q6.2, 1 s
   "Tag_67" : Bool = PLC GRIPPER_UNHOLD AT %Q6.3, 1 s
   "PLUG LIFTING CYLINDER UP(1)" : Bool = PLC "PLUG LIFTING CYLINDER UP(1)" AT %Q6.1, 1 s
   "PLUG LIFTING CYLINDER DOWN" : Bool = PLC "PLUG LIFTING CYLINDER DOWN" AT %M151.3, 1 s
   "PLUG LIFTING CYLINDER FORWARD" : Bool = PLC "PLUG LIFTING CYLINDER FORWARD" AT %M151.4, 1 s
   "PLUG LIFTING CYLINDER REVERSE" : Bool = PLC "PLUG LIFTING CYLINDER REVERSE" AT %M151.5, 1 s
   "TRAY STOPPER UP" : Bool = PLC "TRAY STOPPER UP" AT %M151.6, 1 s
   "TRAY STOPPER DOWN" : Bool = PLC "TRAY STOPPER DOWN" AT %M151.7, 1 s
   "TRAY LATCH UP" : Bool = PLC "TRAY LATCH UP" AT %M152.0, 1 s
   "TRAY LATCH DOWN" : Bool = PLC "TRAY LATCH DOWN" AT %M152.1, 1 s
   "INDIVIDULISER CYLINDER  UP" : Bool = PLC "INDIVIDULISER CYLINDER  UP" AT %M150.2, 1 s
   "INDIVIDULISER CYLINDER DOWN" : Bool = PLC "INDIVIDULISER CYLINDER DOWN" AT %M150.3, 1 s
   "TRAY LIFTING HEIGHT LEVELING UP" : Bool = PLC "TRAY LIFTING HEIGHT LEVELING UP" AT %M150.4, 1 s
   "TRAY LIFTING HEIGHT LEVELING DOWN" : Bool = PLC "TRAY LIFTING HEIGHT LEVELING DOWN" AT %M150.5, 1 s
   "TRAY LIFTING CYLINDER  UP" : Bool = PLC "TRAY LIFTING CYLINDER  UP" AT %M150.6, 1 s
   "TRAY LIFTING CYLINDER  DOWN" : Bool = PLC "TRAY LIFTING CYLINDER  DOWN" AT %M150.7, 1 s
   "TRAY LIFTING CYLINDER FORWARD" : Bool = PLC "TRAY LIFTING CYLINDER FORWARD" AT %M151.0, 1 s
   "TRAY LIFTING CYLINDER REVERSE" : Bool = PLC "TRAY LIFTING CYLINDER REVERSE" AT %M151.1, 1 s
   "MAN WALKER DOWN" : Bool = PLC "MAN WALKER DOWN" AT %M500.1, 1 s
   "MAN WALKER UP" : Bool = PLC "MAN WALKER UP" AT %M500.0, 1 s
   "HMI_TRAY_HEIGHT_DOWN" : Bool = PLC HMI_TRAY_HEIGHT_DOWN AT %M501.0, 1 s
   "HMI_TRAY_HEIGHT_UP" : Bool = PLC HMI_TRAY_HEIGHT_UP AT %M501.1, 1 s
   "HMI_TRAY_LIFT_DOWN" : Bool = PLC HMI_TRAY_LIFT_DOWN AT %M500.6, 1 s
   "HMI_TRAY_LIFT_UP" : Bool = PLC HMI_TRAY_LIFT_UP AT %M500.7, 1 s
   "HMI_TRAY_LIFT_REVERSE" : Bool = PLC HMI_TRAY_LIFT_REVERSE AT %M501.3, 1 s
   "HMI_TRAY_LIFT_FORWARD" : Bool = PLC HMI_TRAY_LIFT_FORWARD AT %M501.2, 1 s
   "HMI_PLUG_LIFT_DOWN" : Bool = PLC HMI_PLUG_LIFT_DOWN AT %M500.3, 1 s
   "HMI_PLUG_LIFT_UP" : Bool = PLC HMI_PLUG_LIFT_UP AT %M500.2, 1 s
   "HMI_PLUG_LIFT_REV" : Bool = PLC HMI_PLUG_LIFT_REV AT %M502.1, 1 s
   "HMI_PLUG_LIFT_FWD" : Bool = PLC HMI_PLUG_LIFT_FWD AT %M502.0, 1 s
   "HMI_GRIPPER_UNHOLD" : Bool = PLC HMI_GRIPPER_UNHOLD AT %M500.5, 1 s
   "HMI_GRIPPER_HOLD" : Bool = PLC HMI_GRIPPER_HOLD AT %M500.4, 1 s
   "PLUG LIFTING CYLINDER UP(2)" : Bool = PLC "PLUG LIFTING CYLINDER UP(1)" AT %Q6.1, 1 s
   "PLUG LIFTING CYLINDER_UP" : Bool = PLC "PLUG LIFTING CYLINDER_UP" AT %I3.4, 1 s
   "PLUG LIFTING CYLINDER_DOWN" : Bool = PLC "PLUG LIFTING CYLINDER_DOWN" AT %I3.3, 1 s
   "PLUG LIFTING CYLINDER_REVERSE" : Bool = PLC "PLUG LIFTING CYLINDER_REVERSE" AT %I3.6, 1 s
   "PLUG LIFTING CYLINDER_FORWARD" : Bool = PLC "PLUG LIFTING CYLINDER_FORWARD" AT %I3.5, 1 s
   "GRIPPER_UNHOLD" : Bool = PLC GRIPPER_UNHOLD AT %Q6.3, 1 s
   "GRIPPER_HOLD" : Bool = PLC GRIPPER_HOLD AT %Q6.2, 1 s
   "INDIVIDULISER_DOWN" : Bool = PLC INDIVIDULISER_DOWN AT %I2.4, 1 s
   "INDIVIDULISER_UP" : Bool = PLC INDIVIDULISER_UP AT %I2.3, 1 s
   "WALKER BEAM UP" : Bool = PLC "WALKER BEAM UP" AT %Q0.0, 1 s
   "WALKER BEAM DOWN" : Bool = PLC "WALKER BEAM DOWN" AT %Q0.1, 1 s
   "TRAY LIFTING DOWN" : Bool = PLC "TRAY LIFTING DOWN" AT %Q6.6, 1 s
   "TRAY PICKUP HEIGHT DOWN" : Bool = PLC "TRAY PICKUP HEIGHT DOWN" AT %Q7.0, 1 s
   "TRAY LIFTING HEIGHT LEVELING_UP" : Bool = PLC "TRAY LIFTING HEIGHT LEVELING_UP" AT %I2.5, 1 s
   "TRAY LIFTING HEIGHT LEVELING_DOWN" : Bool = PLC "TRAY LIFTING HEIGHT LEVELING_DOWN" AT %I2.6, 1 s
   "TRAY PICKUP UP" : Bool = PLC "TRAY PICKUP UP" AT %Q7.1, 1 s
   "TRAY LIFTING CYLINDER _DOWN" : Bool = PLC "TRAY LIFTING CYLINDER _DOWN" AT %I3.0, 1 s
   "TRAY LIFTING CYLINDER  UP_OUTPUT" : Bool = PLC "TRAY LIFTING CYLINDER  UP_OUTPUT" AT %Q6.7, 1 s
   "TRAY LIFTING CYLINDER_FORWARD_RS" : Bool = PLC "TRAY LIFTING CYLINDER_FORWARD_RS" AT %I3.1, 1 s
   "TRAY LIFTING CYLINDER_REVERSE_RS" : Bool = PLC "TRAY LIFTING CYLINDER_REVERSE_RS" AT %I3.2, 1 s
   "TRAY LIFTING FWD_" : Bool = PLC "TRAY LIFTING FWD_" AT %Q7.2, 1 s
   "TRAY_LIFT_REVERSE" : Bool = PLC TRAY_LIFT_REVERSE AT %Q7.3, 1 s
   "PLUG SENSOR MOUNTED ON CHUTE_INPUT" : Bool = PLC "PLUG SENSOR MOUNTED ON CHUTE_INPUT" AT %I1.0, 1 s
   "ALARM_1" : Word = PLC ALARM_1 AT %MW60, 1 s
   "ALL_UNIT_INITIAL" : Bool = PLC ALL_UNIT_INITIAL AT %Q0.2, 1 s
   "TRAY LIFTING CYLINDER _UP" : Bool = PLC "TRAY LIFTING CYLINDER _UP" AT %I2.7, 1 s
   "PLUG_LIFT_DOWN" : Bool = PLC PLUG_LIFT_DOWN AT %Q6.0, 1 s
   "PLUG_LIFT_REV" : Bool = PLC PLUG_LIFT_REV AT %Q6.4, 1 s
   "PLUG_LIFT_FWD" : Bool = PLC PLUG_LIFT_FWD AT %Q6.5, 1 s
   "HMI_TRAY_PRESENT_INITIAL" : Bool = PLC HMI_TRAY_PRESENT_INITIAL AT %M25.2, 1 s

HMI tags "IO MONITOR"
   "0_BIT" : Int, internal
   "1_BIT" : Int, internal
   "2_BIT" : Int, internal
   "3_BIT" : Int, internal
   "4_BIT" : Int, internal
   "5_BIT" : Int, internal
   "6_BIT" : Int, internal
   "7_BIT" : Int, internal
   "BYTE SELECTION" : Int, internal
   "I BIT_0" : Bool AT %I0.0, 1 s
   "I BIT_1" : Bool AT %I0.1, 1 s
   "I BIT_2" : Bool AT %I0.2, 1 s
   "I BIT_3" : Bool AT %I0.3, 1 s
   "I BIT_4" : Bool AT %I0.4, 1 s
   "I BIT_5" : Bool AT %I0.5, 1 s
   "I BIT_6" : Bool AT %I0.6, 1 s
   "I BIT_7" : Bool AT %I0.7, 1 s
   "Q BIT_0" : Bool AT %Q0.0, 1 s
   "Q BIT_1" : Bool AT %Q0.1, 1 s
   "Q BIT_2" : Bool AT %Q0.2, 1 s
   "Q BIT_3" : Bool AT %Q0.3, 1 s
   "Q BIT_4" : Bool AT %Q0.4, 1 s
   "Q BIT_5" : Bool AT %Q0.5, 1 s
   "Q BIT_6" : Bool AT %Q0.6, 1 s
   "Q BIT_7" : Bool AT %Q0.7, 1 s

discrete alarms
   1: 'CONTROL OFF', class Errors, trigger "ALARM_1" bit 0
      on Coming: ActivateScreen("ALARMS", 0)
      on Going: ActivateScreen("MAIN", 0)
   2: 'EMERGENCY PRESSED', class Errors, trigger "ALARM_1" bit 1
      on Coming: ActivateScreen("ALARMS", 0)
      on Going: ActivateScreen("MAIN", 0)
   3: 'TRAY NOT PRESENT', class Errors, trigger "ALARM_1" bit 2
      on Going: ActivateScreen("MAIN", 0)
      on Coming: ActivateScreen("ALARMS", 0)
   4: 'MPCB TRIPPED', class Errors, trigger "ALARM_1" bit 3
      on Coming: ActivateScreen("ALARMS", 0)
      on Going: ActivateScreen("MAIN", 0)
   5: 'AUTO OFF', class Errors, trigger "ALARM_1" bit 4
      on Going: ActivateScreen("MAIN", 0)
      on Coming: ActivateScreen("ALARMS", 0)
   6: 'AIR PRESSURE LOW', class Errors, trigger "ALARM_1" bit 5
      on Coming: ActivateScreen("ALARMS", 0)
      on Going: ActivateScreen("MAIN", 0)
   7: 'WAITING FOR PLUGS FROM SB UNIT', class Errors, trigger "ALARM_1" bit 6
      on Coming: ActivateScreen("ALARMS", 0)
      on Going: ActivateScreen("MAIN", 0)
   8: 'TRAY NOT PRESENT AT BOTTOM CONVEYOR END', class Errors, trigger "ALARM_1" bit 7
      on Coming: ActivateScreen("ALARMS", 0)
      on Going: ActivateScreen("MAIN", 0)

text list "INPUT ADDRESS": 0 'I0.0'; 1 'I0.1'; 2 'I0.2'; 3 'I0.3'; 4 'I0.4'; 5 'I0.5'; 6 'I0.6'; 7 'I0.7'; 8 'I1.0'; 9 'I1.1'; 10 'I1.2'; 11 'I1.3'; 12 'I1.4'; 13 'I1.5'; 14 '-- --'; 15 '-- --'; 16 'I2.0'; 17 'I2.1'; 18 'I2.2'; 19 'I2.3'; 20 'I2.4'; 21 'I2.5'; 22 'I2.6'; 23 'I2.7'; 24 'I3.0'; 25 'I3.1'; 26 'I3.2'; 27 'I3.3'; 28 'I3.4'; 29 'I3.5'; 30 'I3.6'; 31 'I3.7'; 32 'I4.0'; 33 'I4.1'; 34 'I4.2'; 35 'I4.3'; 36 'I4.4'; 37 'I4.5'; 38 'I4.6'; 39 'I4.7'; 40 'I5.0'; 41 'I5.1'; 42 'I5.2'; 43 'I5.3'; 44 'I5.4'; 45 'I5.5'; 46 'I5.6'; 47 'I5.7'

text list "INPUT ADDRESS COMMENT": 0 'CONVEYOR MPCB TRIP FEEDBACK'; 1 'CONTROL ON'; 2 'INITIAL RESET'; 3 'FAULT RESET'; 4 'AUTO MODE'; 5 'MANUAL MODE'; 6 'CYCLE START'; 7 'CYCLE STOP'; 8 'PLUG SENSOR MOUNTED ON CHUTE'; 9 'PNEUMATIC AIR PRESSURE'; 10 'PLUG COUNTING'; 11 'INDIVIDULISER CYL.-1 UP RS'; 12 'INDIVIDULISER CYL.-1 DOWN RS'; 13 'INDIVIDULISER CYL.-2 UP RS'; 14 ''; 15 ''; 16 'INDIVIDULISER CYL.-2 DOWN RS'; 17 'INDIVIDULISER CYL.-3 UP RS'; 18 'INDIVIDULISER CYL.-3 DOWN RS'; 19 'INDIVIDULISER CYL.-4 UP RS'; 20 'INDIVIDULISER CYL.-4 DOWN RS'; 21 'TRAY LIFTING HEIGHT LEVELING UP RS'; 22 'TRAY LIFTING HEIGHT LEVELING DOWN RS'; 23 'TRAY LIFTING CYLINDER UP READ SWITCH'; 24 'TRAY LIFTING CYLINDER DOWN READ SWITCH'; 25 '"TRAY LIFTING CYLINDER FORWARD READ SWITCH"'; 26 '"TRAY LIFTING CYLINDER REVERSE READ SWITCH"'; 27 '"PLUG LIFTING CYLINDER DOWN READ SWITCH"'; 28 '"PLUG LIFTING CYLINDER UP READ SWITCH"'; 29 '"PLUG LIFTING CYLINDER FORWARD READ SWITCH"'; 30 '"PLUG LIFTING CYLINDER REVERSE READ SWITCH"'; 31 '"TRAY STOPPER DOWN READ SWITCH"'; 32 '"TRAY STOPPER UP READ SWITCH"'; 33 'TRAY RIGHT SENSOR'; 34 'SPARE'; 35 'UPPER CONVEYOR RIGHT SENSOR'; 36 'UPPER CONVEYOR LEFT SENSOR'; 37 '"TRAY PRESENT SENSOR-RIGHT PROXIMITY"'; 38 'SPARE'; 39 '"TRAY PRESENT SENSOR-LEFT PROXIMITY"'; 40 'TRAY LEFT SENSOR'; 41 ''; 42 'K1 CONTACTOR FEEDBACK FROM MPCB'; 43 'K2 CONTACTOR FEEDBACK FROM MPCB'; 44 'CONFIRMATION TO START UP/DOWN INDIVIDULISERS'; 45 'DOOR LOCK SWITCH'; 46 ''; 47 ''

text list "INPUT BYTE SELECTION": 0 'IB0'; 1 'IB1'; 2 'IB2'; 3 'IB3'; 4 'IB4'; 5 'IB5'; 6 'IB6'; 7 'IB7'

text list "OUTPUT ADDRESS": 0 'Q0.0'; 1 'Q0.1'; 2 'Q0.2'; 3 'Q0.3'; 4 'Q0.4'; 5 'Q0.5'; 6 'Q0.6'; 7 'Q0.7'; 8 'Q1.0'; 9 'Q1.1'; 10 '--'; 11 '--'; 12 '--'; 13 '--'; 14 '--'; 15 '--'; 16 'Q2.0'; 17 'Q2.1'; 18 'Q2.2'; 19 'Q2.3'; 20 'Q2.4'; 21 'Q2.5'; 22 'Q2.6'; 23 'Q2.7'; 24 'Q3.0'; 25 'Q3.1'; 26 'Q3.2'; 27 'Q3.3'; 28 'Q3.4'; 29 'Q3.5'; 30 'Q3.6'; 31 'Q3.7'; 32 'Q4.0'; 33 'Q4.1'; 34 'Q4.2'; 35 'Q4.3'; 36 'Q4.4'; 37 'Q4.5'; 38 'Q4.6'; 39 'Q4.7'; 40 'Q5.0'; 41 'Q5.1'; 42 'Q5.2'; 43 'Q5.3'; 44 'Q5.4'; 45 'Q5.5'; 46 'Q5.6'; 47 'Q5.7'; 48 'Q6.0'; 49 'Q6.1'; 50 'Q6.2'; 51 'Q6.3'; 52 'Q6.4'; 53 'Q6.5'; 54 'Q6.6'; 55 'Q6.7'; 56 'Q7.0'; 57 'Q7.1'; 58 'Q7.2'; 59 'Q7.3'; 60 'Q7.4'; 61 'Q7.5'; 62 'Q7.6'; 63 'Q7.7'

text list "OUTADDRESS COMMENT": 0 'INDIVIDULISER CYLINDER UP'; 1 'INDIVIDULISER CYLINDER DOWN'; 2 ''; 3 'CYCLE STRT ILPB INDICATOR'; 4 ''; 5 ''; 6 '"BUZZER"'; 7 'CONTROL ON OUTPUT'; 8 '"CONVEYOR -1 RUN OUTPUT"'; 9 '"CONVEYOR 2 RUN OUTPUT"'; 10 '--- ---'; 11 '--- ---'; 12 '--- ---'; 13 '--- ---'; 14 '--- ---'; 15 '--- ---'; 16 'SPARE'; 17 'SPARE'; 18 'SPARE'; 19 'SPARE'; 20 'SPARE'; 21 'SPARE'; 22 'SPARE'; 23 'SPARE'; 24 'SPARE'; 25 'SPARE'; 26 'SPARE'; 27 'SPARE'; 28 'SPARE'; 29 'SPARE'; 30 'SPARE'; 31 'SPARE'; 32 'SPARE'; 33 'SPARE'; 34 'SPARE'; 35 'SPARE'; 36 'SPARE'; 37 'SPARE'; 38 'SPARE'; 39 'SPARE'; 40 'SPARE'; 41 'SPARE'; 42 'SPARE'; 43 '"TOWER LAMP RED"'; 44 '"TOWER LAMP YELLOW"'; 45 '"TOWER LAMP GREEN"'; 46 '"TOWER LAMP BLUE"'; 47 '"TOWER LAMP WHITE"'; 48 '"PLUG LIFTING CYLINDER DOWN"'; 49 '"PLUG LIFTING CYLINDER UP"'; 50 '"PLUG HOLD O/P"'; 51 '"PLUG UNHOLD O/P"'; 52 '"PLUG LIFTING CYLINDER REVERSE"'; 53 '"PLUG LIFTING CYLINDER FORWARD"'; 54 '"TRAY LIFTING CYLINDER DOWN"'; 55 '"TRAY LIFTING CYLINDER UP"'; 56 '"TRAY LIFTING HEIGHT LEVELING DOWN"'; 57 '"TRAY LIFTING HEIGHT LEVELING UP"'; 58 '"TRAY LIFTING CYLINDER FORWARD"'; 59 '"TRAY LIFTING CYLINDER REVERSE"'; 60 '"TRAY LATCH UP"'; 61 '"TRAY LATCH DOWN"'; 62 '"TRAY STOPPER UP"'; 63 '"TRAY STOPPER DOWN"'

text list "OUT BYTE SELECTION": 0 'QB0'; 1 'QB1'; 2 'QB2'; 3 'QB3'; 4 'QB4'; 5 'QB5'; 6 'QB6'; 7 'QB7'

text list "ERROR MESSAGES": 4 'INDIVIDULISER CYL.-2 RS ERROR BOTH ARE NOT SENSED'; 1 'INDIVIDULISER CYL.-1 RS ERROR BOTH ARE SENSED'; 2 'INDIVIDULISER CYL.-1 RS ERROR BOTH ARE NOT SENSED'; 3 'INDIVIDULISER CYL.-2 RS ERROR BOTH ARE SENSED'; 5 'INDIVIDULISER CYL.-3RS ERROR BOTH ARE SENSED'; 6 'INDIVIDULISER CYL.-3 RS ERROR BOTH ARE NOT SENSED'; 7 'INDIVIDULISER CYL.-4 RS ERROR BOTH ARE SENSED'; 8 'INDIVIDULISER CYL.-4 RS ERROR BOTH ARE NOT SENSED'; 9 'TRAY LIFTING HEIGHT LEVELING CYL.UP/DOWN RS ERROR BOTH ARE SENSED'; 10 'TRAY LIFTING HEIGHT LEVELING CYL.UP/DOWN RS ERROR BOTH ARE NOT SENSED'; 11 'TRAY LIFTING CYL.UP/DOWN RS ERROR BOTH ARE SENSED'; 12 'TRAY LIFTING CYL.UP/DOWN RS ERROR BOTH ARE NOT SENSED'; 13 'TRAY LIFTING CYL.FWD/REV RS ERROR BOTH ARE SENSED'; 14 'TRAY LIFTING CYL.FWD/REV RS ERROR BOTH ARE NOT SENSED'; 15 'PLUG LIFTING CYL.UP/DOWN RS ERROR BOTH ARE SENSED'; 16 'PLUG LIFTING CYL.UP/DOWN RS ERROR BOTH ARE NOT SENSED'; 17 'PLUG LIFTING CYL.FWD/REV RS ERROR BOTH ARE SENSED'; 18 'PLUG LIFTING CYL.FWD/REV RS ERROR BOTH ARE NOT SENSED'; 19 'TRAY STOPPER CYL.UP/DOWN RS ERROR BOTH ARE SENSED'; 20 'TRAY STOPPER CYL.UP/DOWN RS ERROR BOTH ARE NOT SENSED'; 21 'TRAY LATCH CYL.UP/DOWN RS ERROR BOTH ARE SENSED'; 22 'TRAY LATCH CYL.UP/DOWN RS ERROR BOTH ARE NOT SENSED'; 23 'PLUG HOLDER ERROR'; 24 'EMERGENCY SWITCH PRESSED'; 25 'MPCB TRIPPED'; 26 'AIR PRESSURE LOW'; 27 ''; 28 ''; 29 ''; 30 ''

screen "HAND_1" 800x480
   Button "Button_1" at 600,420 size 191x57; TextOff 'Next'
      on Click: ActivateScreen("HAND_2", 0)
   Button "Button_2" at 5,420 size 191x57; TextOff 'HOME'
      on Click: ActivateScreen("MAIN", 0)
   TextField "Text field_3" at 203,40 size 406x29; Text 'INDIVIDULISER CYLINDER UP/DWN'
   Button "Button_3" at 30,13 size 65x94; TextOff 'Text'; PictureOn "LEFT_ARROW_ACTIVE"; PictureOff "LEFT_ARR"
      on Press: function_b14e0dd5("MAN WALKER DOWN", 0)
      Appearance <- "MAN WALKER DOWN"
   TextField "Text field_5" at 115,13 size 64x44; Text 'DOWN'
      Appearance <- "INDIVIDULISER_DOWN"
   Button "Button_11" at 97,13 size 11x44; TextOff 'Text'; PictureOff "Untitled_2"
   Button "Button_20" at 687,13 size 11x44; TextOff 'Text'; PictureOff "Untitled_2"
   Button "Button_4" at 700,13 size 65x94; TextOff 'Text'; PictureOn "RIGHT_ARROW_ACTIVE"; PictureOff "RIGHT_ARROW_1"
      on Press: function_b14e0dd5("MAN WALKER UP", 0)
      Appearance <- "MAN WALKER UP"
   TextField "Text field_32" at 115,63 size 64x44; Text 'Q0.1'
      Appearance <- "WALKER BEAM DOWN"
   TextField "Text field_6" at 620,13 size 64x44; Text 'UP'
      Appearance <- "INDIVIDULISER_UP"
   TextField "Text field_33" at 620,63 size 64x44; Text 'Q0.0'
      Appearance <- "WALKER BEAM UP"
   Button "Button_5" at 97,63 size 11x44; TextOff 'Text'; PictureOff "Untitled_2"
   Button "Button_6" at 687,63 size 11x44; TextOff 'Text'; PictureOff "Untitled_2"
   TextField "Text field_4" at 203,128 size 364x29; Text 'TRAY LIFTING HEIGHT LEVELING'
   TextField "Text field_7" at 280,159 size 217x29; Text 'CYLINDER UP/DWN'
   Button "Button_7" at 687,110 size 11x44; TextOff 'Text'; PictureOff "Untitled_2"
      on Press: function_b14e0dd5("TRAY LIFTING HEIGHT LEVELING UP FROM HMI", 0)
   Button "Button_8" at 700,110 size 65x94; TextOff 'Text'; PictureOn "RIGHT_ARROW_ACTIVE"; PictureOff "RIGHT_ARROW_1"
      on Press: function_b14e0dd5("HMI_TRAY_HEIGHT_UP", 0)
      Appearance <- "HMI_TRAY_HEIGHT_UP"
   TextField "Text field_8" at 620,110 size 64x44; Text 'UP'
      Appearance <- "TRAY LIFTING HEIGHT LEVELING_UP"
   TextField "Text field_9" at 620,160 size 64x44; Text 'Q7.1'
      Appearance <- "TRAY PICKUP UP"
   Button "Button_9" at 687,160 size 11x44; TextOff 'Text'; PictureOff "Untitled_2"
   Button "Button_10" at 30,110 size 65x94; TextOff 'Text'; PictureOn "LEFT_ARROW_ACTIVE"; PictureOff "LEFT_ARR"
      on Press: function_b14e0dd5("HMI_TRAY_HEIGHT_DOWN", 0)
      Appearance <- "HMI_TRAY_LIFT_DOWN"
   TextField "Text field_10" at 115,110 size 64x44; Text 'DOWN'
      Appearance <- "TRAY LIFTING HEIGHT LEVELING_DOWN"
   Button "Button_12" at 97,110 size 11x44; TextOff 'Text'; PictureOff "Untitled_2"
   TextField "Text field_11" at 115,160 size 64x44; Text 'Q7.0'
      Appearance <- "TRAY PICKUP HEIGHT DOWN"
   Button "Button_13" at 97,160 size 11x44; TextOff 'Text'; PictureOff "Untitled_2"
   TextField "Text field_1" at 203,234 size 396x29; Text 'TRAY LIFTING CYLINDER UP/DOWN'
   Button "Button_14" at 687,206 size 11x44; TextOff 'Text'; PictureOff "Untitled_2"
   Button "Button_15" at 700,206 size 65x94; TextOff 'Text'; PictureOn "RIGHT_ARROW_ACTIVE"; PictureOff "RIGHT_ARROW_1"
      on Press: function_b14e0dd5("HMI_TRAY_LIFT_UP", 0)
      Appearance <- "HMI_TRAY_LIFT_UP"
   TextField "Text field_14" at 620,206 size 64x44; Text 'UP'
      Appearance <- "TRAY LIFTING CYLINDER _UP"
   TextField "Text field_15" at 620,256 size 64x44; Text 'Q6.7'
      Appearance <- "TRAY LIFTING CYLINDER  UP_OUTPUT"
   Button "Button_16" at 687,256 size 11x44; TextOff 'Text'; PictureOff "Untitled_2"
   Button "Button_17" at 30,206 size 65x94; TextOff 'Text'; PictureOn "LEFT_ARROW_ACTIVE"; PictureOff "LEFT_ARR"
      on Press: function_b14e0dd5("HMI_TRAY_LIFT_DOWN", 0)
      Appearance <- "HMI_TRAY_LIFT_DOWN"
   TextField "Text field_16" at 116,206 size 64x44; Text 'DOWN'
      Appearance <- "TRAY LIFTING CYLINDER _DOWN"
   Button "Button_18" at 98,206 size 11x44; TextOff 'Text'; PictureOff "Untitled_2"
   TextField "Text field_17" at 116,256 size 64x44; Text 'Q6.6'
      Appearance <- "TRAY LIFTING DOWN"
   Button "Button_19" at 98,256 size 11x44; TextOff 'Text'; PictureOff "Untitled_2"
   TextField "Text field_12" at 202,332 size 382x29; Text 'TRAY LIFTING CYLINDER FWD/REV'
   Button "Button_21" at 686,304 size 11x44; TextOff 'Text'; PictureOff "Untitled_2"
   Button "Button_22" at 699,304 size 65x94; TextOff 'Text'; PictureOn "RIGHT_ARROW_ACTIVE"; PictureOff "RIGHT_ARROW_1"
      on Press: function_b14e0dd5("HMI_TRAY_LIFT_FORWARD", 0)
      Appearance <- "HMI_TRAY_LIFT_FORWARD"
   TextField "Text field_13" at 619,304 size 64x44; Text 'FWD'
      Appearance <- "TRAY LIFTING CYLINDER_FORWARD_RS"
   TextField "Text field_18" at 619,354 size 64x44; Text 'Q7.2'
      Appearance <- "TRAY LIFTING FWD_"
   Button "Button_23" at 686,354 size 11x44; TextOff 'Text'; PictureOff "Untitled_2"
   Button "Button_24" at 29,304 size 65x94; TextOff 'Text'; PictureOn "LEFT_ARROW_ACTIVE"; PictureOff "LEFT_ARR"
      on Press: function_b14e0dd5("HMI_TRAY_LIFT_REVERSE", 0)
      Appearance <- "HMI_TRAY_LIFT_REVERSE"
   TextField "Text field_19" at 115,304 size 64x44; Text 'REV'
      Appearance <- "TRAY LIFTING CYLINDER_REVERSE_RS"
   Button "Button_25" at 97,304 size 11x44; TextOff 'Text'; PictureOff "Untitled_2"
   TextField "Text field_20" at 115,354 size 64x44; Text 'Q7.3'
      Appearance <- "TRAY_LIFT_REVERSE"
   Button "Button_26" at 97,354 size 11x44; TextOff 'Text'; PictureOff "Untitled_2"
   Softkey "Softkey_F1" at 0,0 size 0x0
      on KeyDown: ActivateScreen("MAIN", 0)
   Softkey "Softkey_F8" at 0,0 size 0x0
      on KeyDown: ActivateScreen("HAND_2", 0)

screen "HAND_2" 800x480
   TextField "Text field_3" at 181,322 size 22x34; Text 'Text'
   TextField "Text field_4" at 163,356 size 22x34; Text 'Text'
   TextField "Text field_1" at 229,385 size 22x34; Text 'Text'
   TextField "Text field_2" at 242,419 size 22x34; Text 'Text'
   Button "Button_1" at 600,420 size 191x57; TextOff 'Next'
      on Click: ActivateScreen("HAND_3", 0)
   Button "Button_2" at 5,420 size 191x57; TextOff 'BACK'
      on Click: ActivateScreen("HAND_1", 0)
   TextField "Text field_12" at 206,35 size 376x29; Text 'PLUG LIFTING CYLINDER UP/DWN'
   Button "Button_21" at 690,7 size 11x44; TextOff 'Text'; PictureOff "Untitled_2"
      on Press: function_b14e0dd5("PLUG LIFTING CYLINDER UP FROM HMI", 0)
   Button "Button_22" at 703,7 size 65x94; TextOff 'Text'; PictureOn "RIGHT_ARROW_ACTIVE"; PictureOff "RIGHT_ARROW_1"
      on Press: function_b14e0dd5("HMI_PLUG_LIFT_UP", 0)
      Appearance <- "HMI_PLUG_LIFT_UP"
   TextField "Text field_13" at 623,7 size 64x44; Text 'UP'
      Appearance <- "PLUG LIFTING CYLINDER_UP"
   TextField "Text field_18" at 623,57 size 64x44; Text 'Q6.1'
      Appearance <- "PLUG LIFTING CYLINDER UP(2)"
   Button "Button_23" at 690,57 size 11x44; TextOff 'Text'; PictureOff "Untitled_2"
   Button "Button_24" at 33,7 size 65x94; TextOff 'Text'; PictureOn "LEFT_ARROW_ACTIVE"; PictureOff "LEFT_ARR"
      on Press: function_b14e0dd5("HMI_PLUG_LIFT_DOWN", 0)
      Appearance <- "HMI_PLUG_LIFT_DOWN"
   TextField "Text field_19" at 119,7 size 64x44; Text 'DOWN'
      Appearance <- "PLUG LIFTING CYLINDER_DOWN"
   Button "Button_25" at 101,7 size 11x44; TextOff 'Text'; PictureOff "Untitled_2"
   TextField "Text field_20" at 119,57 size 64x44; Text 'Q6.0'
      Appearance <- "PLUG_LIFT_DOWN"
   Button "Button_26" at 101,57 size 11x44; TextOff 'Text'; PictureOff "Untitled_2"
   TextField "Text field_5" at 207,134 size 384x29; Text 'PLUG LIFTING CYLINDER FWD/REV'
   Button "Button_3" at 691,106 size 11x44; TextOff 'Text'; PictureOff "Untitled_2"
   Button "Button_4" at 704,106 size 65x94; TextOff 'Text'; PictureOn "RIGHT_ARROW_ACTIVE"; PictureOff "RIGHT_ARROW_1"
      on Press: function_b14e0dd5("HMI_PLUG_LIFT_FWD", 0)
      Appearance <- "HMI_PLUG_LIFT_FWD"
   TextField "Text field_6" at 624,106 size 64x44; Text 'FWD'
      Appearance <- "PLUG LIFTING CYLINDER_FORWARD"
   TextField "Text field_7" at 624,156 size 64x44; Text 'Q6.5'
      Appearance <- "PLUG_LIFT_FWD"
   Button "Button_5" at 691,156 size 11x44; TextOff 'Text'; PictureOff "Untitled_2"
   Button "Button_6" at 34,106 size 65x94; TextOff 'Text'; PictureOn "LEFT_ARROW_ACTIVE"; PictureOff "LEFT_ARR"
      on Press: function_b14e0dd5("HMI_PLUG_LIFT_REV", 0)
      Appearance <- "HMI_PLUG_LIFT_REV"
   TextField "Text field_8" at 120,106 size 64x44; Text 'REV'
      Appearance <- "PLUG LIFTING CYLINDER_REVERSE"
   Button "Button_7" at 102,106 size 11x44; TextOff 'Text'; PictureOff "Untitled_2"
   TextField "Text field_9" at 120,156 size 64x44; Text 'Q6.4'
      Appearance <- "PLUG_LIFT_REV"
   Button "Button_8" at 102,156 size 11x44; TextOff 'Text'; PictureOff "Untitled_2"
   TextField "Text field_10" at 208,233 size 321x29; Text 'TRAY STOPPER UP/DWN'
   Button "Button_9" at 692,205 size 11x44; TextOff 'Text'; PictureOff "Untitled_2"
   Button "Button_10" at 705,205 size 65x94; TextOff 'Text'; PictureOn "RIGHT_ARROW_ACTIVE"; PictureOff "RIGHT_ARROW_1"
      on Press: function_b14e0dd5("TRAY STOPPER UP FROM HMI", 0)
   TextField "Text field_11" at 625,205 size 64x44; Text 'UP'
   TextField "Text field_14" at 625,255 size 64x44; Text 'Q7.6'
      Appearance <- "TRAY STOPPER UP"
   Button "Button_11" at 692,255 size 11x44; TextOff 'Text'; PictureOff "Untitled_2"
   Button "Button_12" at 35,205 size 65x94; TextOff 'Text'; PictureOn "LEFT_ARROW_ACTIVE"; PictureOff "LEFT_ARR"
      on Press: function_b14e0dd5("TRAY STOPPER DOWN FROM HMI", 0)
   TextField "Text field_15" at 121,205 size 64x44; Text 'DOWN'
   Button "Button_13" at 103,205 size 11x44; TextOff 'Text'; PictureOff "Untitled_2"
   TextField "Text field_16" at 121,255 size 64x44; Text 'Q7.7'
      Appearance <- "TRAY STOPPER DOWN"
   Button "Button_14" at 103,255 size 11x44; TextOff 'Text'; PictureOff "Untitled_2"
   TextField "Text field_17" at 208,333 size 304x29; Text 'TRAY LATCH UP/DWN'
   Button "Button_15" at 692,305 size 11x44; TextOff 'Text'; PictureOff "Untitled_2"
   Button "Button_16" at 705,305 size 65x94; TextOff 'Text'; PictureOn "RIGHT_ARROW_ACTIVE"; PictureOff "RIGHT_ARROW_1"
      on Press: function_b14e0dd5("TRAY LATCH UP FROM HMI", 0)
   TextField "Text field_21" at 625,305 size 64x44; Text 'UP'
   TextField "Text field_22" at 625,355 size 64x44; Text 'Q7.4'
      Appearance <- "TRAY LATCH UP"
   Button "Button_17" at 692,355 size 11x44; TextOff 'Text'; PictureOff "Untitled_2"
   Button "Button_18" at 35,305 size 65x94; TextOff 'Text'; PictureOn "LEFT_ARROW_ACTIVE"; PictureOff "LEFT_ARR"
      on Press: function_b14e0dd5("TRAY LATCH DOWN FROM HMI", 0)
   TextField "Text field_23" at 121,305 size 64x44; Text 'DOWN'
   Button "Button_19" at 103,305 size 11x44; TextOff 'Text'; PictureOff "Untitled_2"
   TextField "Text field_24" at 121,355 size 64x44; Text 'Q7.5'
      Appearance <- "TRAY LATCH DOWN"
   Button "Button_20" at 103,355 size 11x44; TextOff 'Text'; PictureOff "Untitled_2"
   Button "Button_27" at 293,420 size 191x57; TextOff 'HOME'
      on Click: ActivateScreen("MAIN", 0)
   Softkey "Softkey_F1" at 0,0 size 0x0
      on KeyDown: ActivateScreen("HAND_1", 0)
   Softkey "Softkey_F8" at 0,0 size 0x0
      on KeyDown: ActivateScreen("HAND_3", 0)
   Softkey "Softkey_F5" at 0,0 size 0x0
      on KeyDown: ActivateScreen("MAIN", 0)
   Softkey "Softkey_F4" at 0,0 size 0x0
      on KeyDown: ActivateScreen("MAIN", 0)

